C03628=1090.288,180.141,-70.084,176.047,19.774,152.993
C03629=1090.283,179.893,-70.061,176.045,19.773,152.994
C03630=1090.276,179.644,-70.040,176.042,19.772,152.994
C03631=1090.271,179.395,-70.017,176.039,19.771,152.994
C03632=1090.265,179.146,-69.995,176.036,19.769,152.994
C03633=1090.259,178.898,-69.973,176.034,19.768,152.995
C03634=1090.254,178.648,-69.950,176.031,19.767,152.995
C03635=1090.248,178.399,-69.927,176.028,19.766,152.995
C03636=1090.242,178.150,-69.906,176.025,19.765,152.995
C03637=1090.237,177.901,-69.884,176.023,19.764,152.995
C03638=1090.232,177.652,-69.861,176.020,19.763,152.996
C03639=1090.225,177.403,-69.839,176.017,19.762,152.996
C03640=1090.220,177.155,-69.817,176.014,19.761,152.996
C03641=1090.215,176.906,-69.794,176.012,19.760,152.997
C03642=1090.209,176.656,-69.773,176.009,19.759,152.997
C03643=1090.203,176.407,-69.750,176.006,19.758,152.997
C03644=1090.197,176.131,-69.726,176.003,19.756,152.997
C03645=1090.191,175.854,-69.701,176.001,19.755,152.997
C03646=1090.184,175.577,-69.677,175.997,19.753,152.998
C03647=1090.178,175.300,-69.652,175.994,19.752,152.998
C03648=1090.172,175.051,-69.630,175.992,19.751,152.998
C03649=1090.167,174.803,-69.607,175.989,19.750,152.998
C03650=1090.162,174.553,-69.585,175.986,19.749,152.999
C03651=1090.155,174.304,-69.563,175.983,19.748,152.999
C03652=1090.151,174.055,-69.542,175.981,19.747,152.999
C03653=1090.144,173.806,-69.519,175.978,19.746,152.999
C03654=1090.139,173.557,-69.497,175.975,19.745,153.000
C03655=1090.134,173.308,-69.475,175.972,19.744,153.000
C03656=1090.128,173.059,-69.454,175.970,19.742,153.000
C03657=1090.123,172.811,-69.431,175.967,19.741,153.000
C03658=1090.116,172.561,-69.409,175.965,19.740,153.000
C03659=1090.111,172.312,-69.387,175.962,19.739,153.001
C03660=1090.106,172.063,-69.366,175.960,19.738,153.001
C03661=1090.100,171.814,-69.344,175.957,19.737,153.001
C03662=1090.095,171.565,-69.322,175.954,19.736,153.001
C03663=1090.089,171.317,-69.299,175.952,19.734,153.001
C03664=1090.084,171.068,-69.278,175.949,19.733,153.002
C03665=1090.078,170.819,-69.256,175.946,19.732,153.002
C03666=1090.073,170.570,-69.234,175.943,19.731,153.002
C03667=1090.067,170.321,-69.212,175.941,19.730,153.002
C03668=1090.061,170.071,-69.190,175.938,19.729,153.003
C03669=1090.056,169.822,-69.169,175.935,19.728,153.003
C03670=1090.050,169.573,-69.147,175.933,19.726,153.003
C03671=1090.045,169.324,-69.125,175.930,19.725,153.003
C03672=1090.039,169.076,-69.102,175.927,19.724,153.004
C03673=1090.034,168.827,-69.081,175.925,19.722,153.004
C03674=1090.028,168.578,-69.059,175.923,19.722,153.004
C03675=1090.023,168.329,-69.038,175.920,19.720,153.004
C03676=1090.017,168.080,-69.015,175.917,19.719,153.004
C03677=1090.012,167.831,-68.994,175.915,19.718,153.004
C03678=1090.006,167.582,-68.972,175.912,19.717,153.005
C03679=1090.001,167.333,-68.951,175.909,19.716,153.005
C03680=1089.995,167.083,-68.928,175.906,19.715,153.005
C03681=1089.990,166.835,-68.907,175.904,19.713,153.005
C03682=1089.984,166.586,-68.886,175.901,19.712,153.005
C03683=1089.979,166.336,-68.864,175.899,19.711,153.006
C03684=1089.973,166.088,-68.843,175.896,19.710,153.006
C03685=1089.968,165.838,-68.821,175.893,19.708,153.006
C03686=1089.962,165.590,-68.800,175.891,19.707,153.006
C03687=1089.957,165.340,-68.777,175.889,19.707,153.006
C03688=1089.951,165.092,-68.756,175.886,19.705,153.007
C03689=1089.946,164.842,-68.734,175.883,19.704,153.007
C03690=1089.940,164.594,-68.713,175.881,19.702,153.007
C03691=1089.935,164.345,-68.691,175.878,19.701,153.007
C03692=1089.930,164.095,-68.670,175.875,19.700,153.007
C03693=1089.924,163.847,-68.649,175.873,19.699,153.008
C03694=1089.919,163.597,-68.626,175.870,19.697,153.008
C03695=1089.913,163.349,-68.605,175.867,19.696,153.008
C03696=1089.908,163.100,-68.584,175.865,19.695,153.008
C03697=1089.902,162.851,-68.562,175.863,19.694,153.008
C03698=1089.897,162.601,-68.541,175.860,19.693,153.008
C03699=1089.892,162.353,-68.519,175.858,19.692,153.009
C03700=1089.886,162.103,-68.498,175.855,19.690,153.009
C03701=1089.880,161.855,-68.476,175.852,19.689,153.009
C03702=1089.876,161.606,-68.455,175.850,19.688,153.009
C03703=1089.870,161.356,-68.433,175.847,19.687,153.009
C03704=1089.864,161.108,-68.412,175.844,19.685,153.010
C03705=1089.858,160.858,-68.391,175.842,19.684,153.010
C03706=1089.853,160.609,-68.370,175.840,19.683,153.010
C03707=1089.847,160.360,-68.348,175.837,19.682,153.010
C03708=1089.841,160.083,-68.324,175.834,19.680,153.010
C03709=1089.835,159.806,-68.300,175.831,19.679,153.011
C03710=1089.829,159.528,-68.277,175.828,19.678,153.011
C03711=1089.822,159.251,-68.253,175.825,19.677,153.011
C03712=1089.817,159.002,-68.232,175.823,19.675,153.011
C03713=1089.811,158.754,-68.211,175.820,19.674,153.011
C03714=1089.806,158.504,-68.190,175.818,19.673,153.012
C03715=1089.800,158.255,-68.169,175.815,19.672,153.012
C03716=1089.794,158.005,-68.148,175.813,19.671,153.012
C03717=1089.789,157.757,-68.127,175.810,19.670,153.012
C03718=1089.783,157.508,-68.105,175.808,19.668,153.012
C03719=1089.777,157.259,-68.084,175.805,19.667,153.013
C03720=1089.772,157.010,-68.063,175.802,19.666,153.013
C03721=1089.767,156.761,-68.042,175.800,19.664,153.013
C03722=1089.761,156.511,-68.020,175.797,19.663,153.013
C03723=1089.756,156.262,-68.000,175.795,19.662,153.013
C03724=1089.750,156.014,-67.979,175.793,19.661,153.013
C03725=1089.744,155.764,-67.958,175.790,19.660,153.014
C03726=1089.739,155.516,-67.936,175.787,19.658,153.014
C03727=1089.733,155.266,-67.916,175.785,19.657,153.014
C03728=1089.727,155.017,-67.894,175.782,19.656,153.014
C03729=1089.722,154.768,-67.874,175.779,19.655,153.014
C03730=1089.716,154.520,-67.852,175.778,19.654,153.015
C03731=1089.711,154.270,-67.831,175.775,19.653,153.015
C03732=1089.705,154.021,-67.810,175.772,19.651,153.015
C03733=1089.700,153.772,-67.790,175.769,19.650,153.015
C03734=1089.694,153.524,-67.768,175.767,19.649,153.015
C03735=1089.688,153.274,-67.747,175.764,19.648,153.016
C03736=1089.682,153.025,-67.727,175.762,19.647,153.016
C03737=1089.677,152.776,-67.706,175.760,19.646,153.016
C03738=1089.671,152.527,-67.685,175.757,19.644,153.016
C03739=1089.666,152.278,-67.665,175.755,19.642,153.016
C03740=1089.660,152.029,-67.643,175.752,19.641,153.016
C03741=1089.655,151.780,-67.623,175.749,19.640,153.017
C03742=1089.649,151.530,-67.602,175.747,19.639,153.017
C03743=1089.643,151.282,-67.581,175.745,19.638,153.017
C03744=1089.638,151.032,-67.560,175.742,19.636,153.017
C03745=1089.633,150.783,-67.540,175.739,19.635,153.017
C03746=1089.627,150.534,-67.518,175.737,19.634,153.017
C03747=1089.621,150.285,-67.498,175.734,19.633,153.018
C03748=1089.615,150.036,-67.477,175.732,19.632,153.018
C03749=1089.610,149.788,-67.456,175.730,19.630,153.018
C03750=1089.605,149.539,-67.436,175.727,19.629,153.018
C03751=1089.599,149.289,-67.415,175.725,19.628,153.018
C03752=1089.594,149.040,-67.394,175.722,19.626,153.018
C03753=1089.588,148.791,-67.373,175.719,19.625,153.019
C03754=1089.582,148.542,-67.353,175.718,19.624,153.019
C03755=1089.576,148.292,-67.332,175.715,19.623,153.019
C03756=1089.571,148.043,-67.311,175.712,19.622,153.019
C03757=1089.566,147.794,-67.291,175.710,19.620,153.019
C03758=1089.559,147.546,-67.270,175.707,19.619,153.020
C03759=1089.554,147.297,-67.250,175.705,19.618,153.020
C03760=1089.548,147.047,-67.229,175.703,19.616,153.020
C03761=1089.543,146.798,-67.208,175.700,19.615,153.020
C03762=1089.537,146.549,-67.188,175.697,19.614,153.020
C03763=1089.532,146.300,-67.168,175.695,19.613,153.020
C03764=1089.526,146.051,-67.147,175.693,19.612,153.020
C03765=1089.520,145.801,-67.127,175.690,19.610,153.021
C03766=1089.514,145.553,-67.105,175.688,19.609,153.021
C03767=1089.509,145.304,-67.085,175.685,19.608,153.021
C03768=1089.504,145.055,-67.064,175.683,19.606,153.021
C03769=1089.498,144.806,-67.044,175.681,19.606,153.021
C03770=1089.493,144.557,-67.024,175.678,19.604,153.021
C03771=1089.487,144.307,-67.003,175.676,19.603,153.022
C03772=1089.480,144.030,-66.981,175.673,19.601,153.022
C03773=1089.474,143.752,-66.958,175.670,19.600,153.022
C03774=1089.468,143.475,-66.935,175.668,19.599,153.022
C03775=1089.462,143.197,-66.912,175.665,19.597,153.022
C03776=1089.456,142.948,-66.892,175.662,19.596,153.022
C03777=1089.451,142.699,-66.872,175.660,19.594,153.023
C03778=1089.445,142.450,-66.851,175.657,19.593,153.023
C03779=1089.439,142.201,-66.831,175.655,19.591,153.023
C03780=1089.434,141.951,-66.810,175.653,19.591,153.023
C03781=1089.428,141.702,-66.790,175.650,19.589,153.023
C03782=1089.422,141.453,-66.770,175.648,19.588,153.023
C03783=1089.417,141.204,-66.749,175.645,19.586,153.023
C03784=1089.412,140.955,-66.729,175.643,19.585,153.024
C03785=1089.406,140.706,-66.709,175.641,19.584,153.024
C03786=1089.401,140.457,-66.689,175.638,19.583,153.024
C03787=1089.395,140.208,-66.669,175.636,19.581,153.024
C03788=1089.390,139.959,-66.648,175.633,19.580,153.024
C03789=1089.384,139.710,-66.629,175.631,19.579,153.024
C03790=1089.378,139.461,-66.608,175.629,19.578,153.024
C03791=1089.372,139.211,-66.588,175.626,19.576,153.025
C03792=1089.366,138.962,-66.567,175.624,19.575,153.025
C03793=1089.361,138.713,-66.548,175.622,19.574,153.025
C03794=1089.356,138.463,-66.527,175.619,19.573,153.025
C03795=1089.350,138.215,-66.507,175.617,19.571,153.025
C03796=1089.344,137.966,-66.487,175.614,19.570,153.025
C03797=1089.338,137.717,-66.467,175.611,19.568,153.025
C03798=1089.333,137.467,-66.447,175.610,19.567,153.026
C03799=1089.327,137.218,-66.427,175.607,19.566,153.026
C03800=1089.322,136.969,-66.406,175.604,19.564,153.026
C03801=1089.316,136.720,-66.387,175.602,19.563,153.026
C03802=1089.310,136.471,-66.367,175.600,19.562,153.026
C03803=1089.305,136.222,-66.347,175.598,19.560,153.026
C03804=1089.299,135.973,-66.327,175.595,19.559,153.026
C03805=1089.294,135.724,-66.306,175.592,19.558,153.027
C03806=1089.288,135.474,-66.287,175.591,19.557,153.027
C03807=1089.283,135.225,-66.266,175.588,19.555,153.027
C03808=1089.277,134.976,-66.246,175.586,19.554,153.027
C03809=1089.271,134.727,-66.227,175.583,19.552,153.027
C03810=1089.266,134.478,-66.207,175.581,19.551,153.027
C03811=1089.260,134.229,-66.187,175.579,19.550,153.027
C03812=1089.254,133.980,-66.167,175.576,19.548,153.027
C03813=1089.249,133.730,-66.147,175.574,19.547,153.028
C03814=1089.243,133.482,-66.127,175.572,19.546,153.028
C03815=1089.238,133.232,-66.107,175.569,19.545,153.028
C03816=1089.232,132.983,-66.087,175.567,19.543,153.028
C03817=1089.226,132.734,-66.068,175.565,19.542,153.028
C03818=1089.221,132.485,-66.047,175.562,19.541,153.028
C03819=1089.215,132.236,-66.027,175.560,19.539,153.028
C03820=1089.210,131.986,-66.008,175.557,19.537,153.029
C03821=1089.204,131.737,-65.988,175.556,19.536,153.029
C03822=1089.199,131.488,-65.968,175.553,19.535,153.029
C03823=1089.193,131.239,-65.948,175.550,19.534,153.029
C03824=1089.187,130.989,-65.929,175.548,19.532,153.029
C03825=1089.181,130.741,-65.909,175.546,19.531,153.029
C03826=1089.175,130.491,-65.890,175.544,19.530,153.029
C03827=1089.170,130.242,-65.869,175.541,19.528,153.029
C03828=1089.164,129.993,-65.850,175.539,19.527,153.030
C03829=1089.158,129.744,-65.830,175.537,19.526,153.030
C03830=1089.153,129.494,-65.811,175.534,19.524,153.030
C03831=1089.147,129.246,-65.791,175.532,19.523,153.030
C03832=1089.141,128.996,-65.772,175.530,19.522,153.030
C03833=1089.135,128.747,-65.752,175.527,19.521,153.030
C03834=1089.130,128.498,-65.732,175.525,19.519,153.030
C03835=1089.125,128.250,-65.712,175.522,19.518,153.031
C03836=1089.118,127.971,-65.691,175.520,19.516,153.031
C03837=1089.112,127.694,-65.669,175.517,19.515,153.031
C03838=1089.105,127.416,-65.647,175.515,19.513,153.031
C03839=1089.099,127.138,-65.625,175.512,19.512,153.031
C03840=1089.094,126.889,-65.606,175.510,19.511,153.031
C03841=1089.088,126.640,-65.586,175.508,19.509,153.031
C03842=1089.082,126.391,-65.567,175.505,19.507,153.031
C03843=1089.076,126.141,-65.547,175.504,19.506,153.031
C03844=1089.070,125.892,-65.527,175.501,19.505,153.032
C03845=1089.065,125.644,-65.509,175.499,19.503,153.032
C03846=1089.059,125.394,-65.489,175.496,19.502,153.032
C03847=1089.053,125.146,-65.469,175.494,19.501,153.032
C03848=1089.048,124.896,-65.450,175.492,19.499,153.032
C03849=1089.043,124.646,-65.430,175.489,19.498,153.032
C03850=1089.037,124.397,-65.411,175.488,19.497,153.032
C03851=1089.031,124.148,-65.391,175.485,19.495,153.032
C03852=1089.026,123.899,-65.372,175.482,19.494,153.033
C03853=1089.020,123.650,-65.353,175.481,19.493,153.033
C03854=1089.015,123.400,-65.334,175.478,19.491,153.033
C03855=1089.009,123.152,-65.314,175.476,19.489,153.033
C03856=1089.003,122.902,-65.295,175.473,19.488,153.033
C03857=1088.997,122.653,-65.275,175.472,19.487,153.033
C03858=1088.992,122.404,-65.256,175.469,19.485,153.033
C03859=1088.986,122.155,-65.236,175.467,19.484,153.033
C03860=1088.981,121.906,-65.217,175.465,19.483,153.033
C03861=1088.975,121.656,-65.198,175.462,19.481,153.033
C03862=1088.969,121.407,-65.179,175.460,19.480,153.034
C03863=1088.964,121.158,-65.160,175.458,19.479,153.034
C03864=1088.958,120.909,-65.141,175.456,19.477,153.034
C03865=1088.953,120.659,-65.121,175.453,19.475,153.034
C03866=1088.947,120.411,-65.101,175.452,19.474,153.034
C03867=1088.942,120.162,-65.083,175.449,19.472,153.034
C03868=1088.936,119.912,-65.063,175.447,19.471,153.034
C03869=1088.930,119.663,-65.044,175.445,19.470,153.034
C03870=1088.925,119.414,-65.025,175.443,19.468,153.034
C03871=1088.919,119.165,-65.006,175.440,19.466,153.034
C03872=1088.914,118.915,-64.987,175.438,19.465,153.034
C03873=1088.908,118.666,-64.967,175.436,19.464,153.034
C03874=1088.902,118.416,-64.948,175.433,19.462,153.035
C03875=1088.897,118.168,-64.929,175.431,19.460,153.035
C03876=1088.892,117.918,-64.910,175.429,19.459,153.035
C03877=1088.886,117.669,-64.891,175.427,19.458,153.035
C03878=1088.881,117.420,-64.872,175.424,19.456,153.035
C03879=1088.875,117.171,-64.853,175.423,19.455,153.035
C03880=1088.869,116.921,-64.833,175.420,19.453,153.035
C03881=1088.864,116.673,-64.815,175.418,19.452,153.035
C03882=1088.859,116.423,-64.795,175.416,19.451,153.035
C03883=1088.853,116.174,-64.776,175.414,19.449,153.035
C03884=1088.848,115.925,-64.757,175.411,19.447,153.035
C03885=1088.842,115.676,-64.738,175.409,19.446,153.035
C03886=1088.837,115.426,-64.719,175.407,19.445,153.036
C03887=1088.831,115.177,-64.700,175.405,19.443,153.036
C03888=1088.825,114.928,-64.681,175.403,19.442,153.036
C03889=1088.819,114.679,-64.662,175.400,19.440,153.036
C03890=1088.814,114.430,-64.643,175.398,19.438,153.036
C03891=1088.809,114.181,-64.624,175.396,19.437,153.036
C03892=1088.803,113.931,-64.605,175.394,19.435,153.036
C03893=1088.798,113.682,-64.586,175.391,19.434,153.036
C03894=1088.792,113.433,-64.568,175.390,19.432,153.036
C03895=1088.786,113.183,-64.549,175.387,19.431,153.036
C03896=1088.780,112.934,-64.529,175.386,19.430,153.036
C03897=1088.775,112.685,-64.510,175.383,19.428,153.036
C03898=1088.769,112.436,-64.492,175.381,19.426,153.036
C03899=1088.763,112.186,-64.473,175.379,19.425,153.036
C03900=1088.757,111.908,-64.452,175.377,19.424,153.037
C03901=1088.751,111.631,-64.431,175.374,19.422,153.037
C03902=1088.745,111.353,-64.410,175.372,19.420,153.037
C03903=1088.738,111.076,-64.389,175.369,19.419,153.037
C03904=1088.733,110.827,-64.370,175.367,19.417,153.037
C03905=1088.727,110.578,-64.352,175.365,19.416,153.037
C03906=1088.722,110.328,-64.333,175.363,19.414,153.037
C03907=1088.716,110.079,-64.315,175.360,19.413,153.037
C03908=1088.710,109.830,-64.296,175.358,19.412,153.037
C03909=1088.704,109.580,-64.277,175.356,19.410,153.037
C03910=1088.699,109.331,-64.259,175.354,19.408,153.037
C03911=1088.693,109.082,-64.240,175.352,19.407,153.037
C03912=1088.687,108.833,-64.220,175.350,19.405,153.037
C03913=1088.682,108.584,-64.203,175.347,19.403,153.038
C03914=1088.676,108.334,-64.184,175.345,19.402,153.038
C03915=1088.670,108.085,-64.165,175.343,19.400,153.038
C03916=1088.665,107.836,-64.147,175.341,19.399,153.038
C03917=1088.659,107.586,-64.128,175.339,19.398,153.038
C03918=1088.653,107.338,-64.109,175.337,19.396,153.038
C03919=1088.648,107.088,-64.091,175.335,19.395,153.038
C03920=1088.642,106.839,-64.072,175.332,19.393,153.038
C03921=1088.637,106.590,-64.053,175.330,19.391,153.038
C03922=1088.630,106.340,-64.035,175.328,19.390,153.038
C03923=1088.625,106.091,-64.016,175.326,19.388,153.038
C03924=1088.619,105.842,-63.999,175.324,19.387,153.038
C03925=1088.614,105.593,-63.980,175.322,19.386,153.038
C03926=1088.609,105.343,-63.961,175.320,19.384,153.038
C03927=1088.603,105.094,-63.943,175.318,19.383,153.038
C03928=1088.597,104.845,-63.924,175.316,19.381,153.038
C03929=1088.591,104.595,-63.906,175.313,19.379,153.039
C03930=1088.586,104.347,-63.887,175.311,19.378,153.039
C03931=1088.580,104.097,-63.869,175.309,19.376,153.039
C03932=1088.575,103.848,-63.850,175.307,19.375,153.039
C03933=1088.569,103.598,-63.832,175.305,19.373,153.039
C03934=1088.564,103.350,-63.813,175.303,19.371,153.039
C03935=1088.558,103.100,-63.795,175.301,19.370,153.039
C03936=1088.552,102.851,-63.776,175.299,19.368,153.039
C03937=1088.546,102.601,-63.758,175.297,19.367,153.039
C03938=1088.541,102.353,-63.740,175.295,19.365,153.039
C03939=1088.535,102.103,-63.722,175.292,19.364,153.039
C03940=1088.530,101.854,-63.703,175.291,19.362,153.039
C03941=1088.524,101.604,-63.685,175.288,19.361,153.039
C03942=1088.519,101.355,-63.667,175.287,19.359,153.039
C03943=1088.513,101.106,-63.648,175.284,19.358,153.039
C03944=1088.508,100.857,-63.630,175.282,19.356,153.039
C03945=1088.502,100.607,-63.612,175.280,19.355,153.039
C03946=1088.496,100.358,-63.594,175.278,19.353,153.039
C03947=1088.491,100.108,-63.575,175.276,19.352,153.039
C03948=1088.485,99.860,-63.557,175.274,19.350,153.039
C03949=1088.479,99.610,-63.539,175.271,19.348,153.040
C03950=1088.474,99.361,-63.521,175.270,19.347,153.040
C03951=1088.467,99.112,-63.502,175.267,19.345,153.040
C03952=1088.462,98.863,-63.485,175.266,19.344,153.040
C03953=1088.457,98.613,-63.466,175.263,19.342,153.040
C03954=1088.451,98.364,-63.448,175.261,19.341,153.040
C03955=1088.445,98.114,-63.430,175.259,19.339,153.040
C03956=1088.439,97.865,-63.412,175.257,19.337,153.040
C03957=1088.433,97.616,-63.393,175.255,19.336,153.040
C03958=1088.428,97.367,-63.375,175.253,19.334,153.040
C03959=1088.422,97.117,-63.357,175.250,19.332,153.040
C03960=1088.417,96.868,-63.339,175.249,19.331,153.040
C03961=1088.411,96.619,-63.321,175.247,19.329,153.040
C03962=1088.405,96.370,-63.303,175.245,19.328,153.040
C03963=1088.400,96.121,-63.286,175.243,19.326,153.040
C03964=1088.393,95.843,-63.265,175.240,19.324,153.040
C03965=1088.387,95.565,-63.245,175.238,19.323,153.040
C03966=1088.381,95.288,-63.225,175.235,19.321,153.040
C03967=1088.375,95.010,-63.205,175.234,19.319,153.040
C03968=1088.369,94.760,-63.186,175.231,19.318,153.040
C03969=1088.363,94.511,-63.169,175.229,19.316,153.040
C03970=1088.358,94.262,-63.151,175.227,19.315,153.040
C03971=1088.352,94.013,-63.133,175.225,19.313,153.040
C03972=1088.346,93.764,-63.115,175.223,19.312,153.041
C03973=1088.341,93.514,-63.097,175.221,19.310,153.041
C03974=1088.335,93.265,-63.079,175.220,19.308,153.040
C03975=1088.329,93.016,-63.061,175.217,19.307,153.041
C03976=1088.323,92.766,-63.043,175.215,19.305,153.041
C03977=1088.319,92.517,-63.025,175.213,19.303,153.041
C03978=1088.313,92.268,-63.007,175.211,19.301,153.041
C03979=1088.307,92.018,-62.989,175.209,19.300,153.041
C03980=1088.301,91.769,-62.972,175.207,19.298,153.041
C03981=1088.296,91.520,-62.954,175.205,19.297,153.041
C03982=1088.291,91.270,-62.936,175.203,19.295,153.041
C03983=1088.285,91.021,-62.918,175.201,19.293,153.041
C03984=1088.280,90.772,-62.901,175.199,19.292,153.041
C03985=1088.273,90.522,-62.883,175.197,19.290,153.041
C03986=1088.268,90.273,-62.865,175.195,19.289,153.041
C03987=1088.262,90.024,-62.848,175.193,19.287,153.041
C03988=1088.256,89.774,-62.830,175.191,19.286,153.041
C03989=1088.251,89.525,-62.812,175.189,19.284,153.041
C03990=1088.245,89.276,-62.794,175.187,19.282,153.041
C03991=1088.239,89.027,-62.777,175.185,19.281,153.041
C03992=1088.234,88.778,-62.759,175.183,19.279,153.041
C03993=1088.227,88.528,-62.741,175.181,19.278,153.041
C03994=1088.222,88.279,-62.724,175.179,19.276,153.041
C03995=1088.216,88.030,-62.706,175.177,19.274,153.041
C03996=1088.210,87.780,-62.688,175.175,19.273,153.041
C03997=1088.205,87.531,-62.670,175.173,19.271,153.041
C03998=1088.199,87.282,-62.653,175.171,19.269,153.041
C03999=1088.193,87.032,-62.635,175.169,19.268,153.041
C04000=1088.188,86.783,-62.617,175.167,19.266,153.041
C04001=1088.182,86.534,-62.600,175.165,19.264,153.041
C04002=1088.176,86.284,-62.582,175.163,19.263,153.041
C04003=1088.170,86.035,-62.564,175.161,19.261,153.041
C04004=1088.165,85.786,-62.548,175.159,19.259,153.041
C04005=1088.160,85.537,-62.530,175.157,19.258,153.041
C04006=1088.154,85.287,-62.512,175.155,19.256,153.041
C04007=1088.148,85.038,-62.494,175.153,19.254,153.041
C04008=1088.143,84.789,-62.477,175.152,19.253,153.041
C04009=1088.136,84.539,-62.459,175.149,19.251,153.041
C04010=1088.131,84.289,-62.442,175.148,19.250,153.041
C04011=1088.126,84.040,-62.425,175.145,19.248,153.041
C04012=1088.120,83.791,-62.407,175.143,19.246,153.041
C04013=1088.114,83.542,-62.389,175.141,19.245,153.041
C04014=1088.109,83.292,-62.371,175.139,19.243,153.041
C04015=1088.103,83.043,-62.355,175.138,19.241,153.041
C04016=1088.097,82.794,-62.338,175.135,19.239,153.041
C04017=1088.091,82.544,-62.320,175.134,19.238,153.041
C04018=1088.085,82.295,-62.302,175.131,19.236,153.041
C04019=1088.080,82.046,-62.285,175.130,19.234,153.041
C04020=1088.075,81.797,-62.268,175.128,19.232,153.041
C04021=1088.069,81.548,-62.250,175.126,19.231,153.041
C04022=1088.063,81.298,-62.232,175.124,19.229,153.041
C04023=1088.058,81.048,-62.215,175.122,19.228,153.041
C04024=1088.052,80.799,-62.198,175.120,19.226,153.041
C04025=1088.047,80.550,-62.180,175.118,19.224,153.041
C04026=1088.041,80.301,-62.164,175.116,19.222,153.041
C04027=1088.035,80.051,-62.146,175.114,19.221,153.041
C04028=1088.029,79.774,-62.126,175.112,19.219,153.041
C04029=1088.023,79.496,-62.108,175.110,19.217,153.041
C04030=1088.016,79.218,-62.088,175.108,19.215,153.041
C04031=1088.010,78.941,-62.069,175.105,19.213,153.041
C04032=1088.005,78.692,-62.052,175.104,19.212,153.041
C04033=1087.999,78.442,-62.035,175.102,19.210,153.041
C04034=1087.994,78.193,-62.017,175.100,19.209,153.041
C04035=1087.987,77.944,-62.000,175.098,19.206,153.041
C04036=1087.982,77.694,-61.983,175.096,19.205,153.041
C04037=1087.976,77.445,-61.965,175.094,19.203,153.041
C04038=1087.970,77.196,-61.949,175.092,19.201,153.041
C04039=1087.965,76.947,-61.932,175.090,19.199,153.041
C04040=1087.959,76.696,-61.914,175.088,19.198,153.041
C04041=1087.953,76.447,-61.897,175.086,19.196,153.041
C04042=1087.948,76.198,-61.881,175.085,19.195,153.041
C04043=1087.942,75.949,-61.863,175.082,19.193,153.041
C04044=1087.936,75.700,-61.845,175.081,19.191,153.041
C04045=1087.931,75.451,-61.829,175.078,19.190,153.041
C04046=1087.924,75.201,-61.811,175.077,19.188,153.041
C04047=1087.919,74.951,-61.794,175.075,19.186,153.041
C04048=1087.913,74.702,-61.777,175.073,19.185,153.041
C04049=1087.908,74.453,-61.761,175.071,19.183,153.041
C04050=1087.903,74.203,-61.744,175.069,19.181,153.041
C04051=1087.896,73.954,-61.727,175.067,19.179,153.041
C04052=1087.891,73.705,-61.710,175.066,19.178,153.041
C04053=1087.886,73.456,-61.692,175.063,19.176,153.041
C04054=1087.879,73.206,-61.676,175.062,19.174,153.041
C04055=1087.873,72.957,-61.658,175.060,19.172,153.041
C04056=1087.868,72.707,-61.641,175.058,19.171,153.041
C04057=1087.862,72.458,-61.625,175.056,19.169,153.041
C04058=1087.857,72.209,-61.608,175.054,19.167,153.041
C04059=1087.851,71.959,-61.591,175.052,19.165,153.041
C04060=1087.845,71.710,-61.574,175.051,19.164,153.041
C04061=1087.840,71.460,-61.557,175.048,19.162,153.041
C04062=1087.834,71.211,-61.541,175.047,19.160,153.041
C04063=1087.829,70.962,-61.523,175.044,19.159,153.041
C04064=1087.823,70.713,-61.507,175.043,19.157,153.041
C04065=1087.817,70.463,-61.490,175.041,19.155,153.041
C04066=1087.812,70.214,-61.472,175.039,19.154,153.041
C04067=1087.805,69.964,-61.456,175.037,19.152,153.041
C04068=1087.800,69.714,-61.439,175.035,19.150,153.041
C04069=1087.794,69.466,-61.422,175.033,19.148,153.041
C04070=1087.789,69.216,-61.405,175.032,19.147,153.041
C04071=1087.783,68.967,-61.389,175.029,19.144,153.041
C04072=1087.777,68.718,-61.371,175.028,19.143,153.041
C04073=1087.771,68.468,-61.355,175.026,19.141,153.041
C04074=1087.766,68.219,-61.338,175.024,19.139,153.041
C04075=1087.760,67.969,-61.322,175.022,19.137,153.041
C04076=1087.755,67.720,-61.304,175.021,19.136,153.041
C04077=1087.749,67.471,-61.288,175.018,19.134,153.041
C04078=1087.743,67.221,-61.271,175.017,19.133,153.041
C04079=1087.738,66.972,-61.255,175.014,19.131,153.041
C04080=1087.732,66.722,-61.238,175.013,19.129,153.041
C04081=1087.726,66.473,-61.221,175.011,19.127,153.041
C04082=1087.720,66.224,-61.205,175.009,19.126,153.041
C04083=1087.715,65.974,-61.188,175.007,19.124,153.041
C04084=1087.709,65.725,-61.172,175.005,19.122,153.041
C04085=1087.704,65.475,-61.155,175.003,19.120,153.041
C04086=1087.697,65.227,-61.138,175.002,19.119,153.041
C04087=1087.692,64.977,-61.121,174.999,19.116,153.041
C04088=1087.686,64.728,-61.105,174.998,19.115,153.041
C04089=1087.680,64.478,-61.089,174.996,19.113,153.041
C04090=1087.675,64.229,-61.072,174.994,19.111,153.041
C04091=1087.669,63.979,-61.055,174.993,19.110,153.040
C04092=1087.662,63.701,-61.037,174.990,19.108,153.040
C04093=1087.655,63.424,-61.019,174.988,19.106,153.040
C04094=1087.649,63.146,-61.000,174.986,19.104,153.040
C04095=1087.643,62.869,-60.982,174.984,19.102,153.040
C04096=1087.637,62.620,-60.966,174.982,19.100,153.040
C04097=1087.631,62.370,-60.949,174.981,19.099,153.040
C04098=1087.626,62.121,-60.932,174.978,19.097,153.040
C04099=1087.620,61.871,-60.916,174.977,19.095,153.040
C04100=1087.614,61.622,-60.900,174.975,19.093,153.040
C04101=1087.608,61.373,-60.884,174.973,19.092,153.040
C04102=1087.603,61.123,-60.867,174.971,19.090,153.040
C04103=1087.597,60.874,-60.851,174.970,19.088,153.040
C04104=1087.591,60.624,-60.834,174.968,19.086,153.040
C04105=1087.585,60.375,-60.818,174.966,19.084,153.040
C04106=1087.579,60.125,-60.802,174.964,19.083,153.040
C04107=1087.574,59.876,-60.785,174.962,19.081,153.040
C04108=1087.568,59.626,-60.769,174.961,19.079,153.040
C04109=1087.562,59.377,-60.752,174.958,19.077,153.040
C04110=1087.556,59.128,-60.736,174.957,19.076,153.040
C04111=1087.550,58.878,-60.720,174.955,19.074,153.040
C04112=1087.545,58.629,-60.703,174.953,19.072,153.040
C04113=1087.539,58.379,-60.687,174.951,19.070,153.040
C04114=1087.533,58.130,-60.671,174.949,19.069,153.040
C04115=1087.527,57.881,-60.654,174.948,19.067,153.040
C04116=1087.521,57.631,-60.638,174.946,19.065,153.040
C04117=1087.515,57.382,-60.622,174.944,19.064,153.040
C04118=1087.510,57.132,-60.605,174.942,19.061,153.040
C04119=1087.504,56.883,-60.589,174.941,19.060,153.040
C04120=1087.499,56.634,-60.574,174.938,19.058,153.040
C04121=1087.493,56.384,-60.557,174.937,19.056,153.040
C04122=1087.487,56.135,-60.541,174.935,19.054,153.040
C04123=1087.481,55.886,-60.525,174.933,19.053,153.040
C04124=1087.475,55.636,-60.508,174.932,19.051,153.040
C04125=1087.469,55.387,-60.492,174.929,19.049,153.040
C04126=1087.464,55.137,-60.475,174.928,19.048,153.040
C04127=1087.458,54.887,-60.460,174.926,19.046,153.040
C04128=1087.452,54.638,-60.444,174.925,19.044,153.039
C04129=1087.447,54.389,-60.428,174.922,19.042,153.039
C04130=1087.441,54.140,-60.411,174.921,19.040,153.039
C04131=1087.435,53.891,-60.395,174.919,19.038,153.039
C04132=1087.429,53.641,-60.380,174.917,19.037,153.039
C04133=1087.423,53.391,-60.363,174.916,19.035,153.039
C04134=1087.418,53.142,-60.347,174.913,19.033,153.039
C04135=1087.413,52.893,-60.331,174.912,19.031,153.039
C04136=1087.407,52.643,-60.315,174.910,19.029,153.039
C04137=1087.401,52.394,-60.299,174.908,19.027,153.039
C04138=1087.395,52.144,-60.283,174.906,19.025,153.039
C04139=1087.389,51.895,-60.266,174.905,19.024,153.039
C04140=1087.384,51.645,-60.251,174.903,19.022,153.039
C04141=1087.378,51.396,-60.235,174.901,19.020,153.039
C04142=1087.372,51.147,-60.219,174.900,19.019,153.039
C04143=1087.367,50.897,-60.203,174.898,19.016,153.039
C04144=1087.361,50.648,-60.187,174.896,19.015,153.039
C04145=1087.355,50.398,-60.171,174.894,19.013,153.039
C04146=1087.350,50.149,-60.155,174.892,19.011,153.039
C04147=1087.345,49.899,-60.139,174.891,19.010,153.038
C04148=1087.339,49.650,-60.122,174.889,19.007,153.038
C04149=1087.333,49.400,-60.107,174.887,19.005,153.038
C04150=1087.328,49.152,-60.091,174.885,19.003,153.038
C04151=1087.322,48.902,-60.075,174.884,19.002,153.038
C04152=1087.316,48.652,-60.059,174.881,19.000,153.038
C04153=1087.310,48.403,-60.043,174.880,18.998,153.038
C04154=1087.305,48.154,-60.028,174.879,18.996,153.038
C04155=1087.299,47.904,-60.011,174.877,18.994,153.038
C04156=1087.292,47.626,-59.994,174.875,18.993,153.038
C04157=1087.287,47.348,-59.976,174.873,18.991,153.038
C04158=1087.281,47.070,-59.959,174.871,18.988,153.038
C04159=1087.274,46.793,-59.941,174.869,18.986,153.038
C04160=1087.268,46.543,-59.925,174.867,18.985,153.038
C04161=1087.262,46.294,-59.909,174.866,18.982,153.038
C04162=1087.257,46.044,-59.894,174.864,18.980,153.038
C04163=1087.251,45.795,-59.878,174.862,18.979,153.037
C04164=1087.245,45.545,-59.862,174.860,18.977,153.037
C04165=1087.240,45.296,-59.846,174.859,18.975,153.037
C04166=1087.234,45.047,-59.831,174.857,18.973,153.037
C04167=1087.228,44.797,-59.814,174.855,18.971,153.037
C04168=1087.223,44.548,-59.799,174.854,18.969,153.037
C04169=1087.217,44.299,-59.783,174.852,18.967,153.037
C04170=1087.212,44.049,-59.767,174.850,18.966,153.037
C04171=1087.206,43.800,-59.752,174.849,18.964,153.037
C04172=1087.201,43.550,-59.736,174.847,18.962,153.037
C04173=1087.195,43.300,-59.720,174.845,18.960,153.037
C04174=1087.189,43.051,-59.704,174.843,18.958,153.037
C04175=1087.183,42.802,-59.690,174.841,18.956,153.037
C04176=1087.177,42.552,-59.673,174.840,18.955,153.037
C04177=1087.172,42.302,-59.658,174.838,18.952,153.037
C04178=1087.167,42.054,-59.642,174.837,18.951,153.036
C04179=1087.161,41.804,-59.626,174.834,18.949,153.036
C04180=1087.154,41.554,-59.611,174.833,18.947,153.036
C04181=1087.149,41.305,-59.596,174.831,18.946,153.036
C04182=1087.143,41.055,-59.580,174.829,18.943,153.036
C04183=1087.138,40.806,-59.564,174.828,18.942,153.036
C04184=1087.132,40.557,-59.549,174.826,18.940,153.036
C04185=1087.126,40.307,-59.534,174.824,18.938,153.036
C04186=1087.120,40.057,-59.518,174.823,18.936,153.036
C04187=1087.115,39.809,-59.502,174.821,18.934,153.036
C04188=1087.109,39.559,-59.487,174.819,18.932,153.036
C04189=1087.103,39.309,-59.472,174.817,18.930,153.036
C04190=1087.098,39.060,-59.456,174.816,18.928,153.036
C04191=1087.092,38.810,-59.440,174.814,18.927,153.036
C04192=1087.086,38.560,-59.425,174.812,18.925,153.036
C04193=1087.080,38.312,-59.409,174.811,18.923,153.036
C04194=1087.075,38.062,-59.394,174.809,18.921,153.035
C04195=1087.070,37.813,-59.379,174.807,18.919,153.035
C04196=1087.064,37.563,-59.363,174.806,18.918,153.035
C04197=1087.057,37.314,-59.348,174.804,18.916,153.035
C04198=1087.052,37.065,-59.332,174.802,18.914,153.035
C04199=1087.046,36.815,-59.317,174.801,18.912,153.035
C04200=1087.040,36.565,-59.302,174.799,18.910,153.035
C04201=1087.035,36.316,-59.287,174.797,18.908,153.035
C04202=1087.029,36.067,-59.271,174.795,18.906,153.035
C04203=1087.023,35.817,-59.256,174.794,18.904,153.035
C04204=1087.017,35.568,-59.241,174.792,18.903,153.035
C04205=1087.011,35.318,-59.225,174.790,18.901,153.035
C04206=1087.006,35.068,-59.210,174.789,18.899,153.035
C04207=1087.000,34.819,-59.195,174.787,18.897,153.035
C04208=1086.994,34.569,-59.179,174.785,18.895,153.035
C04209=1086.988,34.321,-59.164,174.784,18.894,153.035
C04210=1086.983,34.071,-59.149,174.781,18.892,153.035
C04211=1086.976,33.821,-59.134,174.780,18.890,153.034
C04212=1086.971,33.572,-59.119,174.779,18.888,153.034
C04213=1086.966,33.322,-59.103,174.777,18.886,153.034
C04214=1086.959,33.073,-59.088,174.775,18.884,153.034
C04215=1086.954,32.823,-59.072,174.774,18.882,153.034
C04216=1086.948,32.574,-59.058,174.772,18.880,153.034
C04217=1086.942,32.324,-59.042,174.770,18.879,153.034
C04218=1086.936,32.075,-59.027,174.768,18.876,153.034
C04219=1086.931,31.825,-59.012,174.767,18.875,153.034
C04220=1086.922,31.451,-58.990,174.765,18.872,153.034
C04221=1086.914,31.077,-58.967,174.762,18.869,153.034
C04222=1086.905,30.702,-58.944,174.759,18.866,153.034
C04223=1086.896,30.328,-58.921,174.757,18.863,153.033
C04224=1086.890,30.078,-58.906,174.756,18.862,153.033
C04225=1086.885,29.829,-58.891,174.753,18.860,153.033
C04226=1086.879,29.579,-58.876,174.752,18.858,153.033
C04227=1086.873,29.330,-58.861,174.750,18.856,153.033
C04228=1086.868,29.080,-58.846,174.748,18.854,153.033
C04229=1086.862,28.831,-58.831,174.747,18.852,153.033
C04230=1086.856,28.581,-58.816,174.745,18.850,153.033
C04231=1086.850,28.332,-58.801,174.743,18.849,153.033
C04232=1086.845,28.082,-58.785,174.742,18.847,153.033
C04233=1086.839,27.833,-58.771,174.740,18.844,153.033
C04234=1086.833,27.584,-58.756,174.739,18.843,153.033
C04235=1086.828,27.334,-58.741,174.737,18.841,153.033
C04236=1086.821,27.084,-58.726,174.735,18.839,153.032
C04237=1086.816,26.835,-58.711,174.734,18.837,153.032
C04238=1086.810,26.585,-58.696,174.732,18.836,153.032
C04239=1086.804,26.336,-58.682,174.730,18.833,153.032
C04240=1086.799,26.086,-58.666,174.729,18.832,153.032
C04241=1086.793,25.837,-58.652,174.727,18.830,153.032
C04242=1086.786,25.588,-58.637,174.725,18.828,153.032
C04243=1086.781,25.338,-58.622,174.724,18.826,153.032
C04244=1086.775,25.088,-58.607,174.723,18.825,153.032
C04245=1086.770,24.839,-58.593,174.720,18.822,153.032
C04246=1086.764,24.589,-58.577,174.719,18.820,153.032
C04247=1086.758,24.340,-58.563,174.718,18.819,153.032
C04248=1086.752,24.091,-58.548,174.715,18.817,153.032
C04249=1086.747,23.841,-58.532,174.714,18.815,153.031
C04250=1086.741,23.591,-58.518,174.713,18.813,153.031
C04251=1086.735,23.342,-58.504,174.710,18.811,153.031
C04252=1086.729,23.092,-58.488,174.709,18.809,153.031
C04253=1086.723,22.843,-58.474,174.708,18.808,153.031
C04254=1086.717,22.594,-58.459,174.706,18.806,153.031
C04255=1086.712,22.344,-58.445,174.704,18.804,153.031
C04256=1086.707,22.095,-58.430,174.703,18.802,153.031
C04257=1086.700,21.845,-58.415,174.701,18.800,153.031
C04258=1086.694,21.596,-58.400,174.700,18.798,153.031
C04259=1086.689,21.346,-58.385,174.698,18.796,153.031
C04260=1086.683,21.097,-58.371,174.696,18.794,153.031
C04261=1086.677,20.847,-58.356,174.695,18.792,153.031
C04262=1086.671,20.598,-58.341,174.693,18.791,153.030
C04263=1086.666,20.348,-58.327,174.691,18.789,153.030
C04264=1086.656,19.946,-58.303,174.688,18.786,153.030
C04265=1086.647,19.543,-58.279,174.686,18.783,153.030
C04266=1086.638,19.141,-58.256,174.683,18.779,153.030
C04267=1086.628,18.738,-58.233,174.681,18.776,153.030
C04268=1086.623,18.489,-58.217,174.679,18.775,153.030
C04269=1086.617,18.240,-58.202,174.678,18.773,153.030
C04270=1086.611,17.990,-58.189,174.676,18.771,153.030
C04271=1086.605,17.740,-58.174,174.674,18.769,153.030
C04272=1086.599,17.491,-58.160,174.673,18.768,153.030
C04273=1086.594,17.242,-58.145,174.671,18.765,153.029
C04274=1086.588,16.992,-58.130,174.669,18.764,153.029
C04275=1086.583,16.742,-58.116,174.668,18.761,153.029
C04276=1086.576,16.493,-58.101,174.666,18.759,153.029
C04277=1086.571,16.243,-58.087,174.665,18.758,153.029
C04278=1086.565,15.994,-58.072,174.663,18.756,153.029
C04279=1086.558,15.744,-58.057,174.661,18.754,153.029
C04280=1086.552,15.468,-58.042,174.660,18.752,153.029
C04281=1086.546,15.192,-58.025,174.658,18.750,153.029
C04282=1086.539,14.915,-58.010,174.656,18.748,153.029
C04283=1086.534,14.638,-57.994,174.654,18.746,153.029
C04284=1086.528,14.389,-57.979,174.653,18.744,153.029
C04285=1086.522,14.140,-57.964,174.652,18.742,153.028
C04286=1086.516,13.890,-57.950,174.649,18.740,153.028
C04287=1086.510,13.641,-57.936,174.648,18.738,153.028
C04288=1086.505,13.391,-57.922,174.646,18.737,153.028
C04289=1086.498,13.141,-57.907,174.644,18.734,153.028
C04290=1086.492,12.892,-57.894,174.643,18.733,153.028
C04291=1086.486,12.643,-57.879,174.642,18.731,153.028
C04292=1086.480,12.393,-57.865,174.640,18.729,153.028
C04293=1086.475,12.143,-57.851,174.638,18.727,153.028
C04294=1086.468,11.894,-57.836,174.637,18.726,153.028
C04295=1086.463,11.644,-57.822,174.636,18.724,153.028
C04296=1086.457,11.395,-57.807,174.633,18.721,153.028
C04297=1086.451,11.145,-57.793,174.632,18.720,153.028
C04298=1086.445,10.896,-57.779,174.630,18.718,153.028
C04299=1086.440,10.646,-57.765,174.628,18.716,153.027
C04300=1086.434,10.396,-57.751,174.627,18.714,153.027
C04301=1086.428,10.147,-57.736,174.626,18.713,153.027
C04302=1086.422,9.897,-57.722,174.624,18.711,153.027
C04303=1086.416,9.648,-57.707,174.622,18.709,153.027
C04304=1086.410,9.399,-57.694,174.621,18.707,153.027
C04305=1086.404,9.149,-57.680,174.619,18.705,153.027
C04306=1086.399,8.900,-57.665,174.617,18.703,153.027
C04307=1086.393,8.650,-57.651,174.616,18.701,153.027
C04308=1086.387,8.400,-57.637,174.615,18.699,153.027
C04309=1086.381,8.151,-57.623,174.612,18.697,153.027
C04310=1086.375,7.901,-57.609,174.611,18.696,153.027
C04311=1086.370,7.651,-57.595,174.610,18.694,153.026
C04312=1086.364,7.402,-57.580,174.608,18.692,153.026
C04313=1086.358,7.153,-57.567,174.606,18.690,153.026
C04314=1086.352,6.903,-57.553,174.605,18.688,153.026
C04315=1086.346,6.654,-57.538,174.603,18.687,153.026
C04316=1086.340,6.404,-57.524,174.601,18.685,153.026
C04317=1086.335,6.155,-57.510,174.600,18.682,153.026
C04318=1086.329,5.904,-57.496,174.599,18.681,153.026
C04319=1086.323,5.656,-57.481,174.597,18.679,153.026
C04320=1086.318,5.406,-57.468,174.595,18.677,153.026
C04321=1086.311,5.157,-57.454,174.594,18.675,153.026
C04322=1086.305,4.906,-57.440,174.593,18.673,153.026
C04323=1086.299,4.657,-57.426,174.591,18.672,153.025
C04324=1086.294,4.408,-57.412,174.589,18.670,153.025
C04325=1086.289,4.158,-57.398,174.588,18.668,153.025
C04326=1086.282,3.908,-57.384,174.586,18.666,153.025
C04327=1086.276,3.659,-57.370,174.584,18.664,153.025
C04328=1086.270,3.410,-57.356,174.583,18.662,153.025
C04329=1086.265,3.160,-57.342,174.581,18.660,153.025
C04330=1086.259,2.911,-57.328,174.580,18.659,153.025
C04331=1086.253,2.660,-57.314,174.578,18.656,153.025
C04332=1086.248,2.411,-57.300,174.576,18.655,153.025
C04333=1086.241,2.162,-57.286,174.575,18.653,153.025
C04334=1086.236,1.913,-57.272,174.573,18.651,153.025
C04335=1086.230,1.663,-57.258,174.572,18.649,153.025
C04336=1086.225,1.413,-57.244,174.570,18.647,153.024
C04337=1086.219,1.163,-57.230,174.569,18.645,153.024
C04338=1086.213,0.914,-57.217,174.567,18.643,153.024
C04339=1086.207,0.664,-57.203,174.566,18.641,153.024
C04340=1086.202,0.415,-57.189,174.564,18.640,153.024
C04341=1086.196,0.165,-57.175,174.563,18.638,153.024
C04342=1086.190,-0.084,-57.161,174.561,18.636,153.024
C04343=1086.184,-0.333,-57.147,174.559,18.634,153.024
C04344=1086.178,-0.608,-57.133,174.558,18.632,153.024
C04345=1086.171,-0.882,-57.117,174.556,18.630,153.024
C04346=1086.166,-1.157,-57.102,174.555,18.628,153.024
C04347=1086.159,-1.431,-57.087,174.553,18.625,153.023
C04348=1086.153,-1.681,-57.073,174.551,18.624,153.023
C04349=1086.148,-1.930,-57.059,174.550,18.622,153.023
C04350=1086.143,-2.180,-57.045,174.548,18.620,153.023
C04351=1086.136,-2.430,-57.032,174.546,18.618,153.023
C04352=1086.130,-2.679,-57.018,174.545,18.616,153.023
C04353=1086.125,-2.929,-57.004,174.544,18.615,153.023
C04354=1086.119,-3.179,-56.990,174.542,18.613,153.023
C04355=1086.113,-3.428,-56.977,174.540,18.610,153.023
C04356=1086.108,-3.677,-56.963,174.539,18.609,153.023
C04357=1086.101,-3.927,-56.950,174.537,18.607,153.023
C04358=1086.096,-4.176,-56.936,174.536,18.605,153.022
C04359=1086.089,-4.426,-56.922,174.534,18.603,153.022
C04360=1086.084,-4.676,-56.908,174.533,18.602,153.022
C04361=1086.078,-4.925,-56.894,174.531,18.600,153.022
C04362=1086.072,-5.175,-56.881,174.529,18.598,153.022
C04363=1086.066,-5.424,-56.867,174.528,18.596,153.022
C04364=1086.060,-5.674,-56.854,174.526,18.595,153.022
C04365=1086.055,-5.923,-56.840,174.525,18.592,153.022
C04366=1086.049,-6.172,-56.827,174.523,18.590,153.022
C04367=1086.043,-6.423,-56.813,174.522,18.589,153.022
C04368=1086.037,-6.673,-56.800,174.520,18.587,153.022
C04369=1086.031,-6.922,-56.786,174.519,18.585,153.022
C04370=1086.025,-7.171,-56.773,174.517,18.583,153.022
C04371=1086.019,-7.421,-56.759,174.516,18.581,153.021
C04372=1086.013,-7.670,-56.746,174.514,18.580,153.021
C04373=1086.008,-7.920,-56.732,174.513,18.578,153.021
C04374=1086.001,-8.169,-56.719,174.510,18.576,153.021
C04375=1085.996,-8.419,-56.706,174.509,18.574,153.021
C04376=1085.990,-8.668,-56.692,174.508,18.572,153.021
C04377=1085.984,-8.919,-56.678,174.506,18.571,153.021
C04378=1085.978,-9.168,-56.665,174.504,18.568,153.021
C04379=1085.972,-9.418,-56.651,174.503,18.567,153.021
C04380=1085.966,-9.667,-56.638,174.502,18.565,153.021
C04381=1085.961,-9.917,-56.624,174.500,18.563,153.021
C04382=1085.955,-10.166,-56.611,174.498,18.561,153.021
C04383=1085.949,-10.416,-56.597,174.497,18.559,153.021
C04384=1085.943,-10.665,-56.584,174.496,18.557,153.020
C04385=1085.937,-10.915,-56.572,174.494,18.556,153.020
C04386=1085.932,-11.165,-56.558,174.493,18.554,153.020
C04387=1085.925,-11.414,-56.544,174.491,18.552,153.020
C04388=1085.920,-11.663,-56.531,174.489,18.550,153.020
C04389=1085.914,-11.913,-56.518,174.488,18.549,153.020
C04390=1085.909,-12.163,-56.504,174.487,18.547,153.020
C04391=1085.902,-12.412,-56.491,174.484,18.545,153.020
C04392=1085.897,-12.662,-56.478,174.483,18.543,153.020
C04393=1085.891,-12.912,-56.464,174.482,18.541,153.020
C04394=1085.885,-13.161,-56.451,174.480,18.539,153.020
C04395=1085.879,-13.410,-56.437,174.478,18.537,153.020
C04396=1085.873,-13.660,-56.425,174.477,18.535,153.020
C04397=1085.868,-13.910,-56.411,174.476,18.534,153.020
C04398=1085.862,-14.159,-56.398,174.474,18.532,153.019
C04399=1085.857,-14.409,-56.384,174.473,18.530,153.019
C04400=1085.850,-14.659,-56.371,174.471,18.528,153.019
C04401=1085.844,-14.908,-56.358,174.469,18.527,153.019
C04402=1085.839,-15.158,-56.345,174.468,18.524,153.019
C04403=1085.833,-15.407,-56.332,174.467,18.523,153.019
C04404=1085.827,-15.657,-56.319,174.464,18.521,153.019
C04405=1085.821,-15.907,-56.306,174.463,18.519,153.019
C04406=1085.815,-16.156,-56.292,174.462,18.517,153.019
C04407=1085.809,-16.406,-56.279,174.460,18.516,153.019
C04408=1085.803,-16.679,-56.265,174.458,18.514,153.019
C04409=1085.797,-16.951,-56.251,174.457,18.512,153.019
C04410=1085.790,-17.224,-56.235,174.456,18.510,153.019
C04411=1085.784,-17.497,-56.221,174.453,18.508,153.019
C04412=1085.778,-17.747,-56.209,174.452,18.506,153.018
C04413=1085.771,-17.996,-56.195,174.451,18.504,153.018
C04414=1085.766,-18.246,-56.183,174.449,18.503,153.018
C04415=1085.759,-18.495,-56.170,174.447,18.501,153.018
C04416=1085.754,-18.745,-56.156,174.446,18.499,153.018
C04417=1085.748,-18.995,-56.143,174.444,18.497,153.018
C04418=1085.742,-19.244,-56.131,174.443,18.496,153.018
C04419=1085.736,-19.494,-56.117,174.442,18.494,153.018
C04420=1085.731,-19.744,-56.104,174.440,18.491,153.018
C04421=1085.724,-19.993,-56.091,174.438,18.490,153.018
C04422=1085.719,-20.243,-56.078,174.437,18.488,153.018
C04423=1085.713,-20.492,-56.065,174.435,18.487,153.018
C04424=1085.707,-20.741,-56.053,174.434,18.485,153.018
C04425=1085.701,-20.991,-56.040,174.432,18.483,153.018
C04426=1085.696,-21.241,-56.026,174.430,18.481,153.017
C04427=1085.689,-21.490,-56.013,174.429,18.479,153.017
C04428=1085.683,-21.740,-56.001,174.428,18.478,153.017
C04429=1085.677,-21.989,-55.987,174.426,18.476,153.017
C04430=1085.671,-22.239,-55.975,174.424,18.474,153.017
C04431=1085.666,-22.489,-55.961,174.423,18.472,153.017
C04432=1085.660,-22.739,-55.948,174.422,18.470,153.017
C04433=1085.654,-22.989,-55.936,174.420,18.469,153.017
C04434=1085.648,-23.237,-55.923,174.419,18.467,153.017
C04435=1085.643,-23.487,-55.910,174.417,18.465,153.017
C04436=1085.636,-23.736,-55.897,174.415,18.463,153.017
C04437=1085.631,-23.986,-55.884,174.414,18.462,153.017
C04438=1085.625,-24.236,-55.871,174.413,18.460,153.017
C04439=1085.619,-24.486,-55.858,174.411,18.458,153.016
C04440=1085.613,-24.735,-55.846,174.409,18.456,153.016
C04441=1085.607,-24.985,-55.833,174.408,18.454,153.016
C04442=1085.602,-25.234,-55.820,174.406,18.453,153.016
C04443=1085.596,-25.484,-55.808,174.405,18.451,153.016
C04444=1085.591,-25.734,-55.794,174.404,18.449,153.016
C04445=1085.584,-25.983,-55.781,174.402,18.448,153.016
C04446=1085.578,-26.233,-55.769,174.400,18.446,153.016
C04447=1085.573,-26.483,-55.756,174.399,18.443,153.016
C04448=1085.567,-26.732,-55.743,174.397,18.442,153.016
C04449=1085.561,-26.981,-55.731,174.396,18.440,153.016
C04450=1085.555,-27.231,-55.718,174.395,18.439,153.016
C04451=1085.549,-27.481,-55.705,174.393,18.436,153.016
C04452=1085.543,-27.730,-55.692,174.391,18.435,153.016
C04453=1085.537,-27.980,-55.680,174.390,18.433,153.016
C04454=1085.531,-28.230,-55.667,174.388,18.432,153.016
C04455=1085.526,-28.479,-55.654,174.387,18.430,153.016
C04456=1085.520,-28.729,-55.642,174.385,18.428,153.015
C04457=1085.514,-28.979,-55.629,174.383,18.426,153.015
C04458=1085.508,-29.228,-55.617,174.382,18.424,153.015
C04459=1085.502,-29.478,-55.603,174.381,18.423,153.015
C04460=1085.496,-29.728,-55.591,174.379,18.421,153.015
C04461=1085.489,-29.977,-55.579,174.378,18.420,153.015
C04462=1085.484,-30.226,-55.567,174.376,18.418,153.015
C04463=1085.478,-30.476,-55.554,174.374,18.416,153.015
C04464=1085.472,-30.726,-55.541,174.373,18.414,153.015
C04465=1085.466,-30.975,-55.528,174.372,18.412,153.015
C04466=1085.460,-31.225,-55.516,174.370,18.411,153.015
C04467=1085.454,-31.474,-55.503,174.369,18.409,153.015
C04468=1085.449,-31.724,-55.491,174.368,18.407,153.015
C04469=1085.443,-31.974,-55.478,174.365,18.405,153.015
C04470=1085.436,-32.223,-55.465,174.364,18.404,153.015
C04471=1085.431,-32.473,-55.453,174.362,18.402,153.015
C04472=1085.424,-32.745,-55.439,174.361,18.401,153.015
C04473=1085.418,-33.017,-55.426,174.359,18.398,153.014
C04474=1085.411,-33.289,-55.412,174.358,18.396,153.014
C04475=1085.405,-33.561,-55.398,174.356,18.395,153.014
C04476=1085.399,-33.811,-55.386,174.355,18.393,153.014
C04477=1085.393,-34.060,-55.374,174.353,18.391,153.014
C04478=1085.387,-34.310,-55.361,174.351,18.389,153.014
C04479=1085.382,-34.560,-55.349,174.350,18.388,153.014
C04480=1085.376,-34.809,-55.337,174.349,18.386,153.014
C04481=1085.370,-35.059,-55.324,174.347,18.385,153.014
C04482=1085.364,-35.309,-55.311,174.346,18.383,153.014
C04483=1085.358,-35.558,-55.299,174.344,18.381,153.014
C04484=1085.352,-35.807,-55.287,174.342,18.379,153.014
C04485=1085.346,-36.057,-55.274,174.341,18.377,153.014
C04486=1085.340,-36.306,-55.262,174.339,18.376,153.014
C04487=1085.335,-36.556,-55.249,174.338,18.374,153.014
C04488=1085.329,-36.806,-55.237,174.337,18.373,153.014
C04489=1085.323,-37.056,-55.224,174.335,18.371,153.014
C04490=1085.317,-37.305,-55.212,174.334,18.370,153.014
C04491=1085.311,-37.555,-55.200,174.332,18.367,153.013
C04492=1085.305,-37.805,-55.188,174.330,18.365,153.013
C04493=1085.300,-38.054,-55.175,174.329,18.364,153.013
C04494=1085.294,-38.304,-55.163,174.328,18.362,153.013
C04495=1085.288,-38.554,-55.150,174.326,18.361,153.013
C04496=1085.282,-38.802,-55.139,174.325,18.359,153.013
C04497=1085.276,-39.052,-55.126,174.323,18.358,153.013
C04498=1085.270,-39.302,-55.114,174.321,18.356,153.013
C04499=1085.264,-39.552,-55.102,174.320,18.353,153.013
C04500=1085.258,-39.802,-55.090,174.318,18.352,153.013
C04501=1085.252,-40.051,-55.078,174.317,18.350,153.013
C04502=1085.246,-40.301,-55.066,174.316,18.349,153.013
C04503=1085.240,-40.551,-55.053,174.314,18.347,153.013
C04504=1085.234,-40.800,-55.041,174.313,18.346,153.013
C04505=1085.228,-41.050,-55.029,174.311,18.344,153.013
C04506=1085.222,-41.300,-55.016,174.309,18.342,153.013
C04507=1085.217,-41.549,-55.004,174.308,18.341,153.013
C04508=1085.210,-41.798,-54.992,174.306,18.339,153.013
C04509=1085.204,-42.048,-54.980,174.305,18.337,153.013
C04510=1085.198,-42.299,-54.968,174.303,18.336,153.013
C04511=1085.192,-42.548,-54.956,174.302,18.334,153.013
C04512=1085.186,-42.797,-54.944,174.301,18.333,153.013
C04513=1085.181,-43.047,-54.931,174.299,18.331,153.013
C04514=1085.175,-43.296,-54.919,174.297,18.329,153.013
C04515=1085.169,-43.546,-54.907,174.296,18.328,153.013
C04516=1085.162,-43.796,-54.896,174.294,18.326,153.012
C04517=1085.157,-44.045,-54.884,174.293,18.324,153.012
C04518=1085.151,-44.295,-54.871,174.292,18.322,153.012
C04519=1085.144,-44.545,-54.859,174.290,18.321,153.012
C04520=1085.139,-44.794,-54.847,174.289,18.319,153.012
C04521=1085.133,-45.044,-54.834,174.287,18.318,153.012
C04522=1085.127,-45.293,-54.823,174.286,18.316,153.012
C04523=1085.122,-45.543,-54.811,174.284,18.314,153.012
C04524=1085.115,-45.793,-54.799,174.282,18.313,153.012
C04525=1085.110,-46.042,-54.787,174.281,18.311,153.012
C04526=1085.104,-46.293,-54.775,174.279,18.309,153.012
C04527=1085.097,-46.542,-54.763,174.278,18.308,153.012
C04528=1085.092,-46.791,-54.751,174.277,18.306,153.012
C04529=1085.085,-47.041,-54.739,174.275,18.305,153.012
C04530=1085.080,-47.291,-54.727,174.274,18.303,153.012
C04531=1085.074,-47.540,-54.715,174.272,18.302,153.012
C04532=1085.068,-47.790,-54.703,174.270,18.300,153.012
C04533=1085.063,-48.040,-54.691,174.269,18.298,153.012
C04534=1085.056,-48.290,-54.679,174.267,18.297,153.012
C04535=1085.051,-48.539,-54.667,174.266,18.295,153.012
C04536=1085.044,-48.812,-54.654,174.264,18.293,153.012
C04537=1085.038,-49.083,-54.641,174.263,18.292,153.012
C04538=1085.031,-49.356,-54.628,174.261,18.289,153.011
C04539=1085.025,-49.629,-54.615,174.260,18.288,153.011
C04540=1085.019,-49.878,-54.603,174.258,18.286,153.011
C04541=1085.013,-50.127,-54.591,174.257,18.285,153.011
C04542=1085.007,-50.378,-54.580,174.255,18.283,153.011
C04543=1085.002,-50.627,-54.568,174.254,18.282,153.011
C04544=1084.995,-50.876,-54.556,174.253,18.280,153.011
C04545=1084.989,-51.127,-54.545,174.251,18.279,153.011
C04546=1084.983,-51.376,-54.532,174.249,18.277,153.011
C04547=1084.977,-51.626,-54.521,174.247,18.275,153.011
C04548=1084.971,-51.875,-54.510,174.246,18.274,153.011
C04549=1084.965,-52.125,-54.497,174.244,18.272,153.011
C04550=1084.959,-52.375,-54.486,174.243,18.271,153.011
C04551=1084.953,-52.624,-54.474,174.242,18.269,153.011
C04552=1084.946,-52.874,-54.463,174.240,18.268,153.011
C04553=1084.941,-53.124,-54.450,174.238,18.266,153.011
C04554=1084.934,-53.373,-54.439,174.237,18.265,153.011
C04555=1084.928,-53.623,-54.428,174.236,18.263,153.011
C04556=1084.923,-53.872,-54.415,174.234,18.262,153.011
C04557=1084.916,-54.122,-54.404,174.233,18.260,153.011
C04558=1084.910,-54.372,-54.392,174.231,18.259,153.011
C04559=1084.904,-54.621,-54.381,174.229,18.257,153.011
C04560=1084.898,-54.871,-54.369,174.227,18.256,153.011
C04561=1084.892,-55.121,-54.358,174.226,18.254,153.011
C04562=1084.886,-55.370,-54.346,174.225,18.252,153.011
C04563=1084.881,-55.620,-54.334,174.223,18.251,153.011
C04564=1084.874,-55.870,-54.322,174.222,18.249,153.011
C04565=1084.868,-56.120,-54.311,174.220,18.248,153.011
C04566=1084.862,-56.369,-54.300,174.219,18.246,153.011
C04567=1084.856,-56.619,-54.288,174.217,18.245,153.011
C04568=1084.850,-56.868,-54.276,174.216,18.244,153.011
C04569=1084.844,-57.118,-54.265,174.215,18.242,153.011
C04570=1084.838,-57.367,-54.253,174.213,18.241,153.011
C04571=1084.832,-57.618,-54.242,174.212,18.239,153.011
C04572=1084.826,-57.866,-54.230,174.210,18.237,153.011
C04573=1084.820,-58.117,-54.219,174.209,18.236,153.011
C04574=1084.814,-58.366,-54.208,174.207,18.235,153.011
C04575=1084.808,-58.616,-54.195,174.206,18.233,153.011
C04576=1084.802,-58.866,-54.184,174.204,18.231,153.011
C04577=1084.796,-59.115,-54.172,174.202,18.230,153.011
C04578=1084.790,-59.365,-54.162,174.201,18.228,153.011
C04579=1084.784,-59.615,-54.150,174.199,18.227,153.011
C04580=1084.778,-59.864,-54.138,174.198,18.226,153.011
C04581=1084.772,-60.114,-54.127,174.196,18.224,153.011
C04582=1084.766,-60.363,-54.115,174.195,18.222,153.011
C04583=1084.760,-60.613,-54.104,174.193,18.221,153.011
C04584=1084.754,-60.863,-54.093,174.192,18.219,153.011
C04585=1084.748,-61.113,-54.081,174.190,18.218,153.011
C04586=1084.742,-61.362,-54.070,174.189,18.217,153.011
C04587=1084.736,-61.612,-54.058,174.187,18.215,153.011
C04588=1084.730,-61.861,-54.047,174.186,18.214,153.011
C04589=1084.723,-62.111,-54.036,174.185,18.212,153.011
C04590=1084.718,-62.361,-54.024,174.183,18.211,153.011
C04591=1084.712,-62.610,-54.013,174.182,18.209,153.011
C04592=1084.706,-62.860,-54.001,174.180,18.208,153.011
C04593=1084.700,-63.110,-53.990,174.179,18.206,153.011
C04594=1084.694,-63.359,-53.979,174.177,18.205,153.011
C04595=1084.689,-63.609,-53.967,174.176,18.204,153.011
C04596=1084.682,-63.859,-53.956,174.174,18.202,153.011
C04597=1084.677,-64.109,-53.945,174.173,18.201,153.011
C04598=1084.671,-64.358,-53.933,174.171,18.199,153.011
C04599=1084.664,-64.608,-53.922,174.170,18.198,153.011
C04600=1084.658,-64.881,-53.910,174.168,18.196,153.011
C04601=1084.652,-65.155,-53.898,174.166,18.194,153.011
C04602=1084.645,-65.429,-53.885,174.165,18.193,153.011
C04603=1084.638,-65.703,-53.873,174.163,18.191,153.011
C04604=1084.632,-65.952,-53.861,174.162,18.190,153.011
C04605=1084.627,-66.201,-53.850,174.160,18.188,153.011
C04606=1084.620,-66.451,-53.839,174.159,18.187,153.011
C04607=1084.615,-66.701,-53.828,174.157,18.186,153.011
C04608=1084.609,-66.951,-53.816,174.156,18.184,153.011
C04609=1084.603,-67.200,-53.805,174.155,18.182,153.011
C04610=1084.597,-67.450,-53.794,174.153,18.181,153.011
C04611=1084.591,-67.700,-53.783,174.151,18.179,153.011
C04612=1084.585,-67.950,-53.772,174.149,18.178,153.011
C04613=1084.579,-68.199,-53.761,174.148,18.176,153.011
C04614=1084.573,-68.449,-53.750,174.146,18.175,153.011
C04615=1084.567,-68.698,-53.738,174.145,18.174,153.011
C04616=1084.562,-68.948,-53.727,174.143,18.172,153.011
C04617=1084.556,-69.198,-53.715,174.142,18.171,153.011
C04618=1084.550,-69.448,-53.704,174.140,18.169,153.011
C04619=1084.544,-69.697,-53.694,174.139,18.168,153.011
C04620=1084.538,-69.947,-53.682,174.137,18.166,153.011
C04621=1084.532,-70.197,-53.671,174.136,18.165,153.011
C04622=1084.526,-70.446,-53.661,174.134,18.164,153.011
C04623=1084.520,-70.696,-53.649,174.133,18.162,153.011
C04624=1084.514,-70.945,-53.638,174.132,18.161,153.011
C04625=1084.508,-71.195,-53.627,174.130,18.160,153.011
C04626=1084.503,-71.445,-53.615,174.128,18.158,153.011
C04627=1084.497,-71.695,-53.604,174.127,18.156,153.011
C04628=1084.491,-71.944,-53.593,174.126,18.155,153.011
C04629=1084.485,-72.194,-53.582,174.124,18.154,153.011
C04630=1084.479,-72.444,-53.571,174.123,18.152,153.011
C04631=1084.473,-72.693,-53.560,174.121,18.151,153.011
C04632=1084.468,-72.943,-53.549,174.119,18.150,153.011
C04633=1084.461,-73.193,-53.538,174.118,18.148,153.011
C04634=1084.455,-73.443,-53.527,174.117,18.147,153.011
C04635=1084.450,-73.692,-53.516,174.115,18.146,153.011
C04636=1084.444,-73.942,-53.506,174.114,18.144,153.011
C04637=1084.438,-74.192,-53.494,174.112,18.142,153.011
C04638=1084.432,-74.441,-53.483,174.110,18.141,153.011
C04639=1084.426,-74.691,-53.473,174.109,18.140,153.011
C04640=1084.420,-74.941,-53.461,174.108,18.138,153.011
C04641=1084.414,-75.190,-53.450,174.107,18.138,153.011
C04642=1084.408,-75.440,-53.440,174.105,18.136,153.011
C04643=1084.401,-75.690,-53.429,174.104,18.135,153.011
C04644=1084.396,-75.939,-53.418,174.102,18.134,153.011
C04645=1084.390,-76.189,-53.407,174.101,18.133,153.011
C04646=1084.384,-76.438,-53.396,174.099,18.131,153.011
C04647=1084.378,-76.688,-53.385,174.098,18.129,153.011
C04648=1084.372,-76.938,-53.374,174.096,18.128,153.011
C04649=1084.366,-77.187,-53.363,174.095,18.127,153.011
C04650=1084.359,-77.437,-53.353,174.093,18.126,153.011
C04651=1084.354,-77.687,-53.342,174.092,18.124,153.011
C04652=1084.348,-77.937,-53.332,174.090,18.123,153.011
C04653=1084.342,-78.186,-53.321,174.089,18.122,153.011
C04654=1084.336,-78.437,-53.309,174.087,18.120,153.011
C04655=1084.330,-78.686,-53.299,174.086,18.119,153.011
C04656=1084.324,-78.935,-53.288,174.084,18.118,153.011
C04657=1084.318,-79.185,-53.277,174.082,18.117,153.011
C04658=1084.312,-79.435,-53.266,174.081,18.115,153.011
C04659=1084.306,-79.685,-53.256,174.079,18.114,153.012
C04660=1084.300,-79.935,-53.245,174.078,18.112,153.012
C04661=1084.294,-80.184,-53.235,174.076,18.111,153.012
C04662=1084.288,-80.434,-53.224,174.075,18.110,153.012
C04663=1084.282,-80.683,-53.213,174.073,18.109,153.012
C04664=1084.275,-80.960,-53.201,174.072,18.107,153.012
C04665=1084.268,-81.235,-53.189,174.070,18.106,153.012
C04666=1084.262,-81.511,-53.178,174.069,18.105,153.012
C04667=1084.254,-81.787,-53.166,174.067,18.104,153.012
C04668=1084.249,-82.037,-53.155,174.065,18.102,153.012
C04669=1084.242,-82.286,-53.145,174.064,18.101,153.012
C04670=1084.236,-82.536,-53.134,174.062,18.100,153.012
C04671=1084.230,-82.786,-53.123,174.061,18.098,153.012
C04672=1084.224,-83.035,-53.113,174.059,18.097,153.012
C04673=1084.218,-83.285,-53.103,174.058,18.096,153.012
C04674=1084.212,-83.535,-53.091,174.056,18.095,153.012
C04675=1084.206,-83.784,-53.081,174.054,18.094,153.012
C04676=1084.200,-84.034,-53.070,174.053,18.092,153.012
C04677=1084.194,-84.283,-53.061,174.051,18.091,153.012
C04678=1084.187,-84.534,-53.049,174.050,18.089,153.012
C04679=1084.182,-84.783,-53.038,174.048,18.088,153.012
C04680=1084.175,-85.033,-53.029,174.047,18.087,153.013
C04681=1084.170,-85.282,-53.018,174.046,18.086,153.013
C04682=1084.164,-85.532,-53.007,174.044,18.085,153.013
C04683=1084.157,-85.782,-52.997,174.043,18.084,153.013
C04684=1084.151,-86.032,-52.986,174.041,18.083,153.013
C04685=1084.145,-86.281,-52.976,174.040,18.082,153.013
C04686=1084.139,-86.531,-52.965,174.038,18.080,153.013
C04687=1084.134,-86.781,-52.955,174.037,18.079,153.013
C04688=1084.127,-87.031,-52.944,174.035,18.078,153.013
C04689=1084.121,-87.280,-52.934,174.033,18.077,153.013
C04690=1084.115,-87.530,-52.924,174.032,18.075,153.013
C04691=1084.109,-87.779,-52.913,174.030,18.074,153.013
C04692=1084.103,-88.029,-52.903,174.029,18.073,153.013
C04693=1084.097,-88.279,-52.892,174.028,18.072,153.013
C04694=1084.091,-88.529,-52.881,174.026,18.071,153.013
C04695=1084.084,-88.778,-52.871,174.025,18.070,153.013
C04696=1084.079,-89.028,-52.861,174.023,18.069,153.013
C04697=1084.072,-89.277,-52.851,174.021,18.068,153.014
C04698=1084.067,-89.527,-52.840,174.020,18.066,153.014
C04699=1084.060,-89.777,-52.830,174.018,18.065,153.014
C04700=1084.054,-90.027,-52.819,174.017,18.064,153.014
C04701=1084.049,-90.277,-52.809,174.015,18.062,153.014
C04702=1084.042,-90.526,-52.799,174.014,18.061,153.014
C04703=1084.037,-90.776,-52.788,174.012,18.060,153.014
C04704=1084.030,-91.025,-52.778,174.011,18.059,153.014
C04705=1084.025,-91.275,-52.768,174.010,18.058,153.014
C04706=1084.018,-91.525,-52.758,174.008,18.057,153.014
C04707=1084.012,-91.775,-52.746,174.007,18.056,153.014
C04708=1084.006,-92.025,-52.737,174.005,18.055,153.014
C04709=1084.000,-92.274,-52.726,174.003,18.054,153.014
C04710=1083.994,-92.524,-52.716,174.002,18.052,153.014
C04711=1083.988,-92.773,-52.705,174.000,18.051,153.014
C04712=1083.983,-93.024,-52.695,173.999,18.050,153.014
C04713=1083.976,-93.273,-52.685,173.997,18.049,153.015
C04714=1083.971,-93.523,-52.675,173.996,18.048,153.014
C04715=1083.964,-93.772,-52.665,173.995,18.047,153.015
C04716=1083.959,-94.022,-52.654,173.993,18.046,153.015
C04717=1083.952,-94.272,-52.644,173.991,18.045,153.015
C04718=1083.947,-94.522,-52.634,173.990,18.043,153.015
C04719=1083.940,-94.771,-52.623,173.988,18.042,153.015
C04720=1083.935,-95.021,-52.613,173.987,18.041,153.015
C04721=1083.928,-95.271,-52.603,173.985,18.040,153.015
C04722=1083.923,-95.521,-52.593,173.983,18.039,153.015
C04723=1083.917,-95.770,-52.583,173.983,18.038,153.015
C04724=1083.911,-96.020,-52.572,173.981,18.037,153.015
C04725=1083.905,-96.270,-52.563,173.979,18.036,153.015
C04726=1083.899,-96.519,-52.552,173.978,18.034,153.015
C04727=1083.893,-96.769,-52.542,173.976,18.033,153.015
C04728=1083.886,-97.047,-52.531,173.975,18.032,153.016
C04729=1083.879,-97.325,-52.520,173.973,18.031,153.016
C04730=1083.873,-97.603,-52.508,173.971,18.030,153.016
C04731=1083.866,-97.881,-52.497,173.970,18.029,153.016
C04732=1083.860,-98.131,-52.487,173.968,18.028,153.016
C04733=1083.854,-98.381,-52.477,173.966,18.027,153.016
C04734=1083.847,-98.631,-52.467,173.965,18.026,153.016
C04735=1083.842,-98.881,-52.457,173.963,18.025,153.016
C04736=1083.835,-99.130,-52.446,173.961,18.024,153.016
C04737=1083.829,-99.380,-52.437,173.961,18.022,153.016
C04738=1083.824,-99.630,-52.427,173.959,18.021,153.016
C04739=1083.817,-99.879,-52.416,173.958,18.020,153.016
C04740=1083.811,-100.129,-52.407,173.956,18.019,153.017
C04741=1083.805,-100.379,-52.397,173.954,18.018,153.017
C04742=1083.799,-100.628,-52.386,173.953,18.017,153.017
C04743=1083.793,-100.878,-52.377,173.951,18.016,153.017
C04744=1083.787,-101.128,-52.367,173.950,18.016,153.017
C04745=1083.781,-101.377,-52.356,173.948,18.015,153.017
C04746=1083.775,-101.627,-52.347,173.947,18.014,153.017
C04747=1083.769,-101.877,-52.337,173.945,18.013,153.017
C04748=1083.762,-102.127,-52.328,173.944,18.011,153.017
C04749=1083.757,-102.376,-52.317,173.942,18.010,153.017
C04750=1083.751,-102.626,-52.307,173.941,18.009,153.018
C04751=1083.744,-102.876,-52.298,173.939,18.008,153.018
C04752=1083.738,-103.125,-52.287,173.938,18.007,153.018
C04753=1083.732,-103.375,-52.277,173.936,18.006,153.018
C04754=1083.726,-103.625,-52.267,173.934,18.005,153.018
C04755=1083.719,-103.875,-52.258,173.933,18.004,153.018
C04756=1083.713,-104.124,-52.247,173.932,18.004,153.018
C04757=1083.708,-104.375,-52.237,173.930,18.003,153.018
C04758=1083.701,-104.624,-52.228,173.929,18.002,153.018
C04759=1083.695,-104.874,-52.218,173.927,18.001,153.018
C04760=1083.690,-105.123,-52.209,173.925,18.000,153.019
C04761=1083.684,-105.373,-52.198,173.924,17.999,153.019
C04762=1083.678,-105.622,-52.188,173.923,17.998,153.019
C04763=1083.672,-105.872,-52.179,173.921,17.997,153.019
C04764=1083.665,-106.122,-52.169,173.919,17.996,153.019
C04765=1083.659,-106.372,-52.160,173.918,17.995,153.019
C04766=1083.653,-106.621,-52.149,173.916,17.994,153.019
C04767=1083.647,-106.871,-52.139,173.914,17.993,153.019
C04768=1083.641,-107.121,-52.130,173.914,17.992,153.019
C04769=1083.635,-107.371,-52.120,173.912,17.991,153.020
C04770=1083.629,-107.621,-52.111,173.910,17.990,153.020
C04771=1083.623,-107.870,-52.101,173.909,17.989,153.020
C04772=1083.617,-108.120,-52.090,173.907,17.988,153.020
C04773=1083.611,-108.370,-52.081,173.906,17.988,153.020
C04774=1083.605,-108.619,-52.071,173.904,17.987,153.020
C04775=1083.598,-108.869,-52.061,173.903,17.986,153.020
C04776=1083.592,-109.119,-52.052,173.901,17.985,153.020
C04777=1083.586,-109.369,-52.042,173.899,17.984,153.021
C04778=1083.580,-109.619,-52.033,173.898,17.984,153.021
C04779=1083.574,-109.868,-52.023,173.897,17.983,153.021
C04780=1083.567,-110.118,-52.013,173.895,17.981,153.021
C04781=1083.561,-110.367,-52.003,173.893,17.980,153.021
C04782=1083.555,-110.617,-51.994,173.892,17.979,153.021
C04783=1083.549,-110.867,-51.984,173.891,17.979,153.021
C04784=1083.543,-111.117,-51.974,173.889,17.978,153.021
C04785=1083.537,-111.367,-51.964,173.887,17.977,153.022
C04786=1083.531,-111.617,-51.955,173.885,17.976,153.022
C04787=1083.525,-111.867,-51.945,173.884,17.975,153.022
C04788=1083.519,-112.116,-51.936,173.883,17.975,153.022
C04789=1083.513,-112.365,-51.926,173.881,17.974,153.022
C04790=1083.507,-112.615,-51.917,173.880,17.973,153.022
C04791=1083.501,-112.865,-51.907,173.878,17.972,153.022
C04792=1083.494,-113.139,-51.896,173.876,17.971,153.022
C04793=1083.487,-113.413,-51.886,173.874,17.970,153.023
C04794=1083.481,-113.687,-51.875,173.873,17.969,153.023
C04795=1083.474,-113.962,-51.866,173.871,17.968,153.023
C04796=1083.467,-114.211,-51.856,173.870,17.967,153.023
C04797=1083.462,-114.462,-51.846,173.868,17.967,153.023
C04798=1083.455,-114.711,-51.837,173.867,17.966,153.023
C04799=1083.449,-114.961,-51.827,173.865,17.965,153.023
C04800=1083.443,-115.211,-51.818,173.863,17.964,153.023
C04801=1083.437,-115.460,-51.808,173.862,17.963,153.024
C04802=1083.430,-115.710,-51.799,173.860,17.963,153.024
C04803=1083.425,-115.959,-51.790,173.859,17.962,153.024
C04804=1083.419,-116.209,-51.780,173.857,17.961,153.024
C04805=1083.412,-116.459,-51.770,173.856,17.960,153.024
C04806=1083.406,-116.709,-51.761,173.854,17.960,153.024
C04807=1083.400,-116.958,-51.751,173.853,17.959,153.024
C04808=1083.394,-117.208,-51.742,173.851,17.958,153.025
C04809=1083.388,-117.458,-51.732,173.850,17.957,153.025
C04810=1083.382,-117.708,-51.723,173.848,17.957,153.025
C04811=1083.375,-117.958,-51.713,173.847,17.956,153.025
C04812=1083.370,-118.207,-51.705,173.845,17.955,153.025
C04813=1083.364,-118.457,-51.695,173.844,17.955,153.025
C04814=1083.357,-118.707,-51.686,173.842,17.954,153.025
C04815=1083.351,-118.956,-51.676,173.840,17.952,153.026
C04816=1083.345,-119.206,-51.667,173.839,17.952,153.026
C04817=1083.339,-119.456,-51.657,173.838,17.951,153.026
C04818=1083.332,-119.706,-51.648,173.836,17.950,153.026
C04819=1083.326,-119.956,-51.638,173.834,17.950,153.026
C04820=1083.321,-120.205,-51.630,173.832,17.949,153.026
C04821=1083.315,-120.455,-51.620,173.832,17.948,153.026
C04822=1083.309,-120.705,-51.611,173.830,17.948,153.027
C04823=1083.302,-120.954,-51.602,173.828,17.947,153.027
C04824=1083.296,-121.204,-51.592,173.826,17.946,153.027
C04825=1083.289,-121.454,-51.582,173.825,17.946,153.027
C04826=1083.284,-121.704,-51.574,173.824,17.945,153.027
C04827=1083.278,-121.954,-51.564,173.822,17.944,153.027
C04828=1083.272,-122.203,-51.555,173.820,17.943,153.028
C04829=1083.265,-122.453,-51.546,173.819,17.943,153.028
C04830=1083.259,-122.703,-51.536,173.817,17.942,153.028
C04831=1083.253,-122.953,-51.527,173.815,17.941,153.028
C04832=1083.247,-123.202,-51.518,173.814,17.940,153.028
C04833=1083.241,-123.452,-51.509,173.813,17.940,153.028
C04834=1083.235,-123.702,-51.499,173.811,17.939,153.029
C04835=1083.228,-123.952,-51.491,173.809,17.938,153.029
C04836=1083.222,-124.202,-51.481,173.807,17.938,153.029
C04837=1083.217,-124.451,-51.472,173.807,17.937,153.029
C04838=1083.210,-124.701,-51.463,173.805,17.936,153.029
C04839=1083.205,-124.951,-51.454,173.803,17.935,153.029
C04840=1083.198,-125.200,-51.445,173.802,17.935,153.030
C04841=1083.191,-125.450,-51.435,173.800,17.934,153.030
C04842=1083.185,-125.700,-51.426,173.799,17.933,153.030
C04843=1083.179,-125.949,-51.418,173.797,17.933,153.030
C04844=1083.173,-126.199,-51.408,173.796,17.932,153.030
C04845=1083.167,-126.449,-51.399,173.794,17.932,153.030
C04846=1083.161,-126.699,-51.390,173.792,17.931,153.031
C04847=1083.154,-126.949,-51.381,173.791,17.931,153.031
C04848=1083.149,-127.198,-51.372,173.789,17.930,153.031
C04849=1083.142,-127.448,-51.362,173.787,17.929,153.031
C04850=1083.136,-127.698,-51.354,173.786,17.928,153.031
C04851=1083.130,-127.948,-51.344,173.785,17.928,153.031
C04852=1083.125,-128.205,-51.335,173.783,17.927,153.032
C04853=1083.124,-128.460,-51.324,173.782,17.925,153.031
C04854=1083.128,-128.715,-51.311,173.782,17.921,153.031
C04855=1083.136,-128.967,-51.297,173.782,17.917,153.030
C04856=1082.735,-128.989,-51.433,173.737,18.034,153.060
C04857=1082.727,-128.736,-51.447,173.738,18.039,153.061
C04858=1082.724,-128.481,-51.459,173.739,18.042,153.061
C04859=1082.724,-128.226,-51.470,173.740,18.044,153.062
C04860=1082.728,-127.970,-51.481,173.740,18.045,153.062
C04861=1082.735,-127.720,-51.490,173.742,18.046,153.061
C04862=1082.740,-127.471,-51.498,173.744,18.047,153.061
C04863=1082.747,-127.221,-51.508,173.746,18.047,153.061
C04864=1082.754,-126.971,-51.517,173.747,18.048,153.061
C04865=1082.759,-126.721,-51.526,173.749,18.048,153.061
C04866=1082.766,-126.471,-51.535,173.750,18.050,153.061
C04867=1082.771,-126.222,-51.544,173.751,18.049,153.060
C04868=1082.778,-125.972,-51.553,173.753,18.051,153.060
C04869=1082.784,-125.722,-51.562,173.755,18.051,153.060
C04870=1082.790,-125.472,-51.572,173.757,18.052,153.060
C04871=1082.797,-125.223,-51.581,173.757,18.053,153.060
C04872=1082.803,-124.972,-51.590,173.759,18.053,153.060
C04873=1082.808,-124.723,-51.599,173.761,18.054,153.059
C04874=1082.815,-124.473,-51.608,173.762,18.054,153.059
C04875=1082.822,-124.224,-51.617,173.764,18.055,153.059
C04876=1082.827,-123.974,-51.626,173.766,18.056,153.059
C04877=1082.834,-123.724,-51.636,173.767,18.057,153.059
C04878=1082.839,-123.475,-51.645,173.768,18.057,153.059
C04879=1082.845,-123.225,-51.654,173.770,18.058,153.058
C04880=1082.851,-122.974,-51.663,173.772,18.059,153.058
C04881=1082.858,-122.725,-51.672,173.774,18.060,153.058
C04882=1082.864,-122.475,-51.682,173.775,18.060,153.058
C04883=1082.870,-122.226,-51.691,173.776,18.061,153.058
C04884=1082.876,-121.976,-51.701,173.778,18.062,153.058
C04885=1082.882,-121.726,-51.709,173.780,18.062,153.058
C04886=1082.888,-121.476,-51.719,173.781,18.063,153.057
C04887=1082.895,-121.227,-51.728,173.782,18.064,153.057
C04888=1082.901,-120.977,-51.738,173.784,18.064,153.057
C04889=1082.907,-120.727,-51.747,173.786,18.065,153.057
C04890=1082.913,-120.477,-51.756,173.787,18.066,153.057
C04891=1082.919,-120.227,-51.765,173.789,18.066,153.057
C04892=1082.925,-119.978,-51.775,173.791,18.067,153.057
C04893=1082.931,-119.728,-51.784,173.792,18.068,153.056
C04894=1082.937,-119.478,-51.794,173.793,18.069,153.056
C04895=1082.944,-119.229,-51.803,173.795,18.069,153.056
C04896=1082.950,-118.979,-51.812,173.797,18.070,153.056
C04897=1082.956,-118.730,-51.822,173.798,18.072,153.056
C04898=1082.962,-118.479,-51.830,173.799,18.072,153.056
C04899=1082.968,-118.229,-51.840,173.801,18.073,153.055
C04900=1082.974,-117.980,-51.850,173.803,18.074,153.055
C04901=1082.980,-117.730,-51.859,173.804,18.075,153.055
C04902=1082.986,-117.480,-51.869,173.806,18.075,153.055
C04903=1082.993,-117.230,-51.878,173.807,18.076,153.055
C04904=1082.999,-116.980,-51.888,173.809,18.077,153.055
C04905=1083.004,-116.731,-51.897,173.811,18.078,153.055
C04906=1083.011,-116.482,-51.907,173.813,18.078,153.054
C04907=1083.017,-116.232,-51.916,173.813,18.079,153.054
C04908=1083.024,-115.982,-51.925,173.815,18.080,153.054
C04909=1083.030,-115.732,-51.935,173.817,18.081,153.054
C04910=1083.036,-115.483,-51.944,173.818,18.082,153.054
C04911=1083.042,-115.232,-51.953,173.819,18.082,153.054
C04912=1083.048,-114.982,-51.963,173.821,18.083,153.054
C04913=1083.054,-114.733,-51.972,173.823,18.084,153.054
C04914=1083.060,-114.483,-51.982,173.824,18.085,153.053
C04915=1083.066,-114.234,-51.991,173.826,18.086,153.053
C04916=1083.072,-113.984,-52.001,173.827,18.086,153.053
C04917=1083.079,-113.709,-52.012,173.829,18.087,153.053
C04918=1083.086,-113.435,-52.022,173.831,18.088,153.053
C04919=1083.093,-113.161,-52.033,173.832,18.089,153.053
C04920=1083.099,-112.886,-52.043,173.834,18.090,153.053
C04921=1083.105,-112.637,-52.053,173.836,18.091,153.053
C04922=1083.111,-112.387,-52.062,173.837,18.092,153.052
C04923=1083.118,-112.137,-52.072,173.839,18.093,153.052
C04924=1083.124,-111.887,-52.082,173.840,18.093,153.052
C04925=1083.130,-111.637,-52.091,173.842,18.094,153.052
C04926=1083.136,-111.388,-52.101,173.843,18.095,153.052
C04927=1083.142,-111.138,-52.110,173.845,18.096,153.052
C04928=1083.148,-110.888,-52.120,173.847,18.097,153.052
C04929=1083.154,-110.638,-52.130,173.848,18.098,153.052
C04930=1083.159,-110.389,-52.139,173.849,18.099,153.051
C04931=1083.166,-110.140,-52.149,173.851,18.100,153.051
C04932=1083.172,-109.890,-52.159,173.853,18.101,153.051
C04933=1083.178,-109.640,-52.169,173.854,18.102,153.051
C04934=1083.184,-109.390,-52.178,173.855,18.102,153.051
C04935=1083.191,-109.140,-52.188,173.857,18.103,153.051
C04936=1083.197,-108.891,-52.197,173.859,18.104,153.051
C04937=1083.203,-108.641,-52.207,173.860,18.105,153.051
C04938=1083.209,-108.391,-52.216,173.862,18.106,153.050
C04939=1083.215,-108.141,-52.226,173.864,18.107,153.050
C04940=1083.221,-107.892,-52.237,173.865,18.108,153.050
C04941=1083.227,-107.642,-52.246,173.866,18.109,153.050
C04942=1083.233,-107.392,-52.256,173.868,18.110,153.050
C04943=1083.239,-107.142,-52.266,173.870,18.111,153.050
C04944=1083.246,-106.892,-52.275,173.871,18.112,153.050
C04945=1083.252,-106.643,-52.285,173.872,18.112,153.050
C04946=1083.258,-106.393,-52.296,173.874,18.113,153.050
C04947=1083.264,-106.143,-52.305,173.875,18.114,153.050
C04948=1083.270,-105.894,-52.315,173.877,18.115,153.049
C04949=1083.276,-105.644,-52.324,173.879,18.116,153.049
C04950=1083.282,-105.394,-52.334,173.881,18.117,153.049
C04951=1083.288,-105.145,-52.345,173.881,18.118,153.049
C04952=1083.294,-104.895,-52.354,173.883,18.119,153.049
C04953=1083.300,-104.645,-52.364,173.885,18.120,153.049
C04954=1083.307,-104.395,-52.373,173.886,18.121,153.049
C04955=1083.312,-104.145,-52.384,173.888,18.123,153.049
C04956=1083.318,-103.896,-52.394,173.889,18.124,153.049
C04957=1083.325,-103.646,-52.403,173.890,18.124,153.049
C04958=1083.331,-103.396,-52.413,173.892,18.125,153.049
C04959=1083.336,-103.146,-52.423,173.894,18.126,153.048
C04960=1083.343,-102.897,-52.433,173.895,18.127,153.048
C04961=1083.349,-102.647,-52.443,173.897,18.128,153.048
C04962=1083.355,-102.397,-52.453,173.899,18.129,153.048
C04963=1083.361,-102.148,-52.463,173.900,18.130,153.048
C04964=1083.367,-101.898,-52.473,173.901,18.131,153.048
C04965=1083.373,-101.648,-52.483,173.903,18.132,153.048
C04966=1083.379,-101.398,-52.492,173.904,18.133,153.048
C04967=1083.385,-101.149,-52.503,173.906,18.134,153.048
C04968=1083.391,-100.899,-52.513,173.908,18.135,153.048
C04969=1083.397,-100.649,-52.522,173.909,18.136,153.047
C04970=1083.403,-100.400,-52.533,173.911,18.137,153.047
C04971=1083.409,-100.150,-52.543,173.912,18.138,153.047
C04972=1083.415,-99.900,-52.552,173.913,18.139,153.047
C04973=1083.423,-99.650,-52.563,173.915,18.140,153.047
C04974=1083.428,-99.400,-52.573,173.917,18.142,153.047
C04975=1083.434,-99.151,-52.583,173.918,18.143,153.047
C04976=1083.441,-98.901,-52.593,173.920,18.144,153.047
C04977=1083.446,-98.651,-52.603,173.922,18.145,153.047
C04978=1083.453,-98.402,-52.613,173.922,18.145,153.047
C04979=1083.459,-98.152,-52.623,173.924,18.146,153.047
C04980=1083.464,-97.902,-52.633,173.925,18.148,153.047
C04981=1083.471,-97.625,-52.644,173.927,18.149,153.046
C04982=1083.478,-97.347,-52.656,173.929,18.150,153.046
C04983=1083.485,-97.068,-52.667,173.931,18.151,153.046
C04984=1083.492,-96.790,-52.679,173.932,18.152,153.046
C04985=1083.497,-96.540,-52.689,173.934,18.153,153.046
C04986=1083.503,-96.290,-52.698,173.935,18.155,153.046
C04987=1083.509,-96.040,-52.709,173.937,18.156,153.046
C04988=1083.515,-95.790,-52.719,173.938,18.157,153.046
C04989=1083.521,-95.541,-52.730,173.940,18.158,153.046
C04990=1083.527,-95.291,-52.739,173.942,18.159,153.046
C04991=1083.533,-95.042,-52.750,173.943,18.161,153.046
C04992=1083.539,-94.792,-52.760,173.945,18.162,153.046
C04993=1083.545,-94.542,-52.770,173.946,18.162,153.046
C04994=1083.551,-94.293,-52.780,173.947,18.163,153.045
C04995=1083.557,-94.043,-52.791,173.949,18.165,153.045
C04996=1083.563,-93.793,-52.800,173.950,18.166,153.045
C04997=1083.569,-93.543,-52.812,173.952,18.167,153.045
C04998=1083.575,-93.293,-52.821,173.953,18.168,153.045
C04999=1083.581,-93.044,-52.832,173.955,18.170,153.045
C05000=1083.587,-92.794,-52.842,173.957,18.171,153.045
C05001=1083.593,-92.545,-52.853,173.958,18.172,153.045
C05002=1083.599,-92.295,-52.862,173.960,18.173,153.045
C05003=1083.605,-92.045,-52.873,173.961,18.174,153.045
C05004=1083.611,-91.795,-52.883,173.962,18.175,153.045
C05005=1083.617,-91.546,-52.893,173.964,18.176,153.045
C05006=1083.624,-91.295,-52.903,173.966,18.177,153.045
C05007=1083.629,-91.046,-52.914,173.967,18.179,153.045
C05008=1083.635,-90.796,-52.924,173.969,18.180,153.045
C05009=1083.641,-90.547,-52.935,173.970,18.181,153.045
C05010=1083.647,-90.297,-52.946,173.972,18.182,153.045
C05011=1083.653,-90.047,-52.955,173.973,18.183,153.044
C05012=1083.659,-89.798,-52.966,173.975,18.185,153.044
C05013=1083.666,-89.547,-52.976,173.976,18.186,153.044
C05014=1083.671,-89.298,-52.987,173.977,18.187,153.044
C05015=1083.678,-89.049,-52.997,173.979,18.188,153.044
C05016=1083.683,-88.799,-53.007,173.980,18.189,153.044
C05017=1083.689,-88.549,-53.018,173.982,18.190,153.044
C05018=1083.695,-88.300,-53.028,173.983,18.192,153.044
C05019=1083.702,-88.049,-53.039,173.985,18.193,153.044
C05020=1083.708,-87.800,-53.049,173.987,18.194,153.044
C05021=1083.713,-87.550,-53.059,173.988,18.195,153.044
C05022=1083.719,-87.300,-53.070,173.990,18.196,153.044
C05023=1083.726,-87.051,-53.081,173.991,18.198,153.044
C05024=1083.731,-86.801,-53.091,173.993,18.199,153.044
C05025=1083.738,-86.551,-53.101,173.994,18.201,153.044
C05026=1083.744,-86.302,-53.112,173.995,18.201,153.044
C05027=1083.750,-86.053,-53.123,173.997,18.202,153.044
C05028=1083.756,-85.802,-53.133,173.998,18.204,153.044
C05029=1083.762,-85.553,-53.144,174.000,18.205,153.044
C05030=1083.769,-85.303,-53.154,174.001,18.206,153.044
C05031=1083.774,-85.053,-53.164,174.003,18.207,153.043
C05032=1083.780,-84.803,-53.175,174.005,18.208,153.043
C05033=1083.786,-84.554,-53.186,174.006,18.210,153.043
C05034=1083.793,-84.304,-53.197,174.008,18.211,153.043
C05035=1083.799,-84.054,-53.206,174.009,18.212,153.043
C05036=1083.805,-83.805,-53.217,174.011,18.213,153.043
C05037=1083.810,-83.555,-53.228,174.012,18.215,153.043
C05038=1083.817,-83.305,-53.239,174.014,18.216,153.043
C05039=1083.823,-83.055,-53.249,174.015,18.218,153.043
C05040=1083.829,-82.806,-53.260,174.017,18.219,153.043
C05041=1083.835,-82.557,-53.270,174.019,18.220,153.043
C05042=1083.841,-82.306,-53.281,174.019,18.221,153.043
C05043=1083.847,-82.057,-53.292,174.021,18.222,153.043
C05044=1083.853,-81.807,-53.302,174.022,18.223,153.043
C05045=1083.860,-81.532,-53.314,174.024,18.224,153.043
C05046=1083.867,-81.255,-53.326,174.026,18.226,153.043
C05047=1083.873,-80.979,-53.338,174.028,18.227,153.043
C05048=1083.880,-80.704,-53.350,174.029,18.229,153.043
C05049=1083.887,-80.454,-53.360,174.031,18.230,153.043
C05050=1083.893,-80.204,-53.370,174.033,18.232,153.043
C05051=1083.898,-79.954,-53.381,174.034,18.233,153.043
C05052=1083.904,-79.705,-53.392,174.036,18.234,153.043
C05053=1083.911,-79.455,-53.403,174.037,18.236,153.043
C05054=1083.917,-79.205,-53.414,174.039,18.237,153.042
C05055=1083.923,-78.956,-53.425,174.040,18.238,153.043
C05056=1083.928,-78.706,-53.435,174.042,18.239,153.042
C05057=1083.935,-78.456,-53.447,174.043,18.241,153.042
C05058=1083.940,-78.206,-53.457,174.045,18.242,153.042
C05059=1083.947,-77.957,-53.467,174.046,18.243,153.042
C05060=1083.953,-77.707,-53.478,174.048,18.245,153.042
C05061=1083.959,-77.457,-53.489,174.049,18.246,153.042
C05062=1083.964,-77.208,-53.500,174.050,18.247,153.042
C05063=1083.970,-76.958,-53.511,174.052,18.248,153.042
C05064=1083.977,-76.708,-53.522,174.053,18.250,153.042
C05065=1083.983,-76.459,-53.533,174.055,18.251,153.042
C05066=1083.989,-76.209,-53.543,174.056,18.252,153.042
C05067=1083.995,-75.959,-53.555,174.058,18.254,153.042
C05068=1084.001,-75.710,-53.566,174.059,18.255,153.042
C05069=1084.007,-75.460,-53.576,174.061,18.256,153.042
C05070=1084.012,-75.211,-53.587,174.062,18.258,153.042
C05071=1084.019,-74.961,-53.599,174.064,18.259,153.042
C05072=1084.024,-74.711,-53.609,174.065,18.261,153.042
C05073=1084.031,-74.462,-53.620,174.067,18.262,153.042
C05074=1084.037,-74.212,-53.631,174.068,18.263,153.042
C05075=1084.043,-73.962,-53.642,174.070,18.265,153.042
C05076=1084.049,-73.713,-53.653,174.071,18.266,153.042
C05077=1084.055,-73.462,-53.664,174.073,18.268,153.042
C05078=1084.061,-73.213,-53.675,174.074,18.269,153.042
C05079=1084.066,-72.963,-53.686,174.076,18.270,153.042
C05080=1084.071,-72.714,-53.697,174.077,18.272,153.042
C05081=1084.078,-72.464,-53.708,174.079,18.273,153.042
C05082=1084.084,-72.214,-53.719,174.080,18.274,153.042
C05083=1084.089,-71.965,-53.730,174.082,18.276,153.042
C05084=1084.096,-71.714,-53.741,174.083,18.278,153.042
C05085=1084.101,-71.465,-53.752,174.084,18.279,153.042
C05086=1084.107,-71.215,-53.763,174.086,18.280,153.042
C05087=1084.113,-70.966,-53.774,174.087,18.282,153.042
C05088=1084.119,-70.716,-53.785,174.089,18.283,153.042
C05089=1084.125,-70.466,-53.796,174.090,18.285,153.042
C05090=1084.131,-70.217,-53.807,174.092,18.286,153.042
C05091=1084.137,-69.967,-53.818,174.093,18.287,153.042
C05092=1084.142,-69.717,-53.830,174.095,18.289,153.042
C05093=1084.148,-69.468,-53.841,174.096,18.291,153.042
C05094=1084.154,-69.218,-53.853,174.098,18.292,153.042
C05095=1084.160,-68.968,-53.863,174.099,18.293,153.042
C05096=1084.166,-68.719,-53.874,174.101,18.295,153.042
C05097=1084.172,-68.468,-53.886,174.102,18.296,153.042
C05098=1084.178,-68.219,-53.896,174.104,18.298,153.042
C05099=1084.184,-67.970,-53.908,174.105,18.299,153.042
C05100=1084.190,-67.720,-53.919,174.107,18.300,153.042
C05101=1084.195,-67.470,-53.931,174.108,18.302,153.042
C05102=1084.201,-67.221,-53.942,174.109,18.303,153.042
C05103=1084.207,-66.970,-53.953,174.111,18.305,153.042
C05104=1084.213,-66.721,-53.964,174.113,18.306,153.042
C05105=1084.220,-66.471,-53.976,174.114,18.308,153.042
C05106=1084.226,-66.222,-53.987,174.116,18.310,153.042
C05107=1084.231,-65.972,-53.997,174.118,18.311,153.042
C05108=1084.237,-65.722,-54.009,174.119,18.313,153.042
C05109=1084.243,-65.448,-54.022,174.121,18.314,153.042
C05110=1084.250,-65.175,-54.034,174.122,18.316,153.042
C05111=1084.257,-64.901,-54.046,174.124,18.317,153.042
C05112=1084.264,-64.628,-54.059,174.125,18.318,153.042
C05113=1084.269,-64.378,-54.070,174.127,18.321,153.042
C05114=1084.275,-64.128,-54.081,174.129,18.322,153.042
C05115=1084.281,-63.878,-54.092,174.130,18.324,153.042
C05116=1084.287,-63.629,-54.104,174.132,18.325,153.042
C05117=1084.293,-63.379,-54.115,174.133,18.327,153.042
C05118=1084.300,-63.129,-54.126,174.135,18.328,153.042
C05119=1084.305,-62.880,-54.139,174.136,18.329,153.042
C05120=1084.311,-62.630,-54.149,174.137,18.331,153.042
C05121=1084.317,-62.380,-54.161,174.139,18.332,153.042
C05122=1084.323,-62.131,-54.172,174.140,18.334,153.042
C05123=1084.329,-61.881,-54.184,174.142,18.336,153.042
C05124=1084.334,-61.631,-54.195,174.143,18.337,153.042
C05125=1084.341,-61.382,-54.207,174.145,18.338,153.042
C05126=1084.347,-61.132,-54.218,174.146,18.340,153.042
C05127=1084.353,-60.882,-54.229,174.148,18.341,153.042
C05128=1084.359,-60.633,-54.241,174.149,18.343,153.042
C05129=1084.365,-60.383,-54.252,174.150,18.344,153.042
C05130=1084.370,-60.133,-54.263,174.152,18.346,153.042
C05131=1084.377,-59.884,-54.275,174.154,18.347,153.042
C05132=1084.383,-59.634,-54.286,174.155,18.348,153.042
C05133=1084.389,-59.384,-54.297,174.156,18.350,153.042
C05134=1084.394,-59.135,-54.310,174.158,18.352,153.042
C05135=1084.401,-58.884,-54.321,174.159,18.353,153.042
C05136=1084.407,-58.636,-54.332,174.161,18.355,153.042
C05137=1084.413,-58.385,-54.344,174.163,18.357,153.043
C05138=1084.419,-58.136,-54.356,174.164,18.358,153.043
C05139=1084.425,-57.886,-54.367,174.166,18.360,153.043
C05140=1084.431,-57.637,-54.378,174.167,18.361,153.042
C05141=1084.437,-57.387,-54.390,174.169,18.362,153.043
C05142=1084.442,-57.137,-54.401,174.170,18.364,153.043
C05143=1084.449,-56.888,-54.413,174.172,18.365,153.043
C05144=1084.455,-56.638,-54.424,174.173,18.367,153.043
C05145=1084.461,-56.389,-54.436,174.175,18.369,153.043
C05146=1084.466,-56.139,-54.448,174.176,18.370,153.043
C05147=1084.473,-55.889,-54.460,174.177,18.372,153.043
C05148=1084.479,-55.639,-54.471,174.179,18.373,153.043
C05149=1084.485,-55.390,-54.483,174.180,18.374,153.043
C05150=1084.491,-55.140,-54.494,174.182,18.376,153.043
C05151=1084.497,-54.891,-54.506,174.183,18.377,153.043
C05152=1084.503,-54.641,-54.517,174.186,18.379,153.043
C05153=1084.509,-54.391,-54.529,174.187,18.381,153.043
C05154=1084.515,-54.141,-54.541,174.188,18.383,153.043
C05155=1084.522,-53.892,-54.553,174.190,18.384,153.043
C05156=1084.528,-53.643,-54.564,174.191,18.386,153.043
C05157=1084.533,-53.392,-54.576,174.193,18.387,153.043
C05158=1084.539,-53.143,-54.588,174.194,18.389,153.043
C05159=1084.546,-52.893,-54.599,174.195,18.390,153.043
C05160=1084.552,-52.643,-54.611,174.197,18.392,153.043
C05161=1084.557,-52.394,-54.622,174.199,18.393,153.043
C05162=1084.564,-52.144,-54.634,174.200,18.394,153.043
C05163=1084.570,-51.895,-54.646,174.201,18.396,153.043
C05164=1084.576,-51.645,-54.658,174.203,18.398,153.043
C05165=1084.582,-51.395,-54.670,174.205,18.400,153.043
C05166=1084.588,-51.146,-54.681,174.207,18.401,153.043
C05167=1084.594,-50.896,-54.693,174.208,18.403,153.043
C05168=1084.601,-50.646,-54.705,174.209,18.404,153.043
C05169=1084.606,-50.397,-54.716,174.211,18.406,153.043
C05170=1084.612,-50.147,-54.728,174.212,18.407,153.043
C05171=1084.617,-49.898,-54.741,174.214,18.409,153.043
C05172=1084.624,-49.648,-54.752,174.215,18.410,153.043
C05173=1084.631,-49.375,-54.766,174.216,18.412,153.043
C05174=1084.637,-49.103,-54.778,174.218,18.415,153.043
C05175=1084.643,-48.830,-54.791,174.220,18.416,153.043
C05176=1084.650,-48.558,-54.804,174.221,18.418,153.043
C05177=1084.655,-48.308,-54.816,174.223,18.419,153.044
C05178=1084.661,-48.059,-54.828,174.224,18.421,153.044
C05179=1084.667,-47.809,-54.840,174.226,18.423,153.044
C05180=1084.673,-47.560,-54.851,174.228,18.424,153.044
C05181=1084.679,-47.310,-54.864,174.229,18.426,153.044
C05182=1084.685,-47.060,-54.876,174.231,18.427,153.044
C05183=1084.691,-46.811,-54.888,174.232,18.429,153.044
C05184=1084.696,-46.560,-54.900,174.233,18.431,153.044
C05185=1084.703,-46.311,-54.912,174.235,18.433,153.044
C05186=1084.708,-46.062,-54.924,174.236,18.434,153.044
C05187=1084.714,-45.812,-54.936,174.237,18.436,153.044
C05188=1084.720,-45.562,-54.947,174.240,18.438,153.044
C05189=1084.726,-45.312,-54.960,174.241,18.439,153.044
C05190=1084.733,-45.063,-54.972,174.243,18.441,153.044
C05191=1084.738,-44.814,-54.984,174.244,18.442,153.044
C05192=1084.744,-44.564,-54.997,174.245,18.444,153.044
C05193=1084.750,-44.314,-55.008,174.247,18.446,153.044
C05194=1084.755,-44.064,-55.020,174.248,18.447,153.044
C05195=1084.762,-43.815,-55.032,174.249,18.449,153.044
C05196=1084.768,-43.565,-55.045,174.251,18.451,153.044
C05197=1084.773,-43.316,-55.057,174.253,18.453,153.044
C05198=1084.780,-43.066,-55.068,174.255,18.454,153.044
C05199=1084.786,-42.816,-55.080,174.256,18.456,153.044
C05200=1084.791,-42.567,-55.093,174.257,18.457,153.045
C05201=1084.798,-42.317,-55.105,174.259,18.459,153.045
C05202=1084.803,-42.067,-55.117,174.260,18.460,153.045
C05203=1084.809,-41.818,-55.129,174.262,18.462,153.045
C05204=1084.815,-41.568,-55.141,174.263,18.464,153.045
C05205=1084.821,-41.318,-55.154,174.265,18.466,153.045
C05206=1084.826,-41.069,-55.165,174.267,18.468,153.045
C05207=1084.833,-40.819,-55.177,174.268,18.469,153.045
C05208=1084.839,-40.569,-55.190,174.269,18.471,153.045
C05209=1084.845,-40.320,-55.202,174.271,18.472,153.045
C05210=1084.851,-40.070,-55.214,174.272,18.474,153.045
C05211=1084.857,-39.821,-55.227,174.274,18.475,153.045
C05212=1084.863,-39.571,-55.239,174.275,18.477,153.045
C05213=1084.869,-39.321,-55.251,174.277,18.480,153.045
C05214=1084.875,-39.072,-55.263,174.278,18.481,153.045
C05215=1084.880,-38.822,-55.276,174.280,18.483,153.045
C05216=1084.887,-38.572,-55.288,174.281,18.484,153.045
C05217=1084.892,-38.323,-55.300,174.283,18.486,153.045
C05218=1084.898,-38.073,-55.313,174.284,18.487,153.045
C05219=1084.904,-37.824,-55.325,174.285,18.489,153.046
C05220=1084.910,-37.574,-55.338,174.288,18.491,153.046
C05221=1084.916,-37.325,-55.349,174.289,18.493,153.046
C05222=1084.922,-37.075,-55.362,174.290,18.495,153.046
C05223=1084.928,-36.825,-55.374,174.292,18.496,153.046
C05224=1084.933,-36.576,-55.387,174.293,18.498,153.046
C05225=1084.939,-36.326,-55.399,174.294,18.500,153.046
C05226=1084.945,-36.076,-55.412,174.296,18.501,153.046
C05227=1084.951,-35.826,-55.424,174.298,18.503,153.046
C05228=1084.957,-35.577,-55.436,174.300,18.505,153.046
C05229=1084.963,-35.327,-55.448,174.301,18.507,153.046
C05230=1084.969,-35.078,-55.461,174.302,18.508,153.046
C05231=1084.975,-34.828,-55.473,174.304,18.510,153.046
C05232=1084.980,-34.578,-55.486,174.305,18.512,153.046
C05233=1084.986,-34.329,-55.498,174.306,18.514,153.046
C05234=1084.992,-34.079,-55.511,174.308,18.516,153.046
C05235=1084.998,-33.829,-55.524,174.310,18.517,153.047
C05236=1085.004,-33.581,-55.536,174.311,18.519,153.047
C05237=1085.010,-33.308,-55.550,174.312,18.521,153.047
C05238=1085.017,-33.036,-55.563,174.315,18.523,153.047
C05239=1085.024,-32.764,-55.577,174.316,18.524,153.047
C05240=1085.029,-32.492,-55.591,174.317,18.526,153.047
C05241=1085.036,-32.242,-55.603,174.319,18.528,153.047
C05242=1085.042,-31.992,-55.615,174.321,18.530,153.047
C05243=1085.048,-31.743,-55.628,174.322,18.532,153.047
C05244=1085.054,-31.493,-55.640,174.324,18.533,153.047
C05245=1085.059,-31.244,-55.652,174.325,18.535,153.047
C05246=1085.065,-30.994,-55.666,174.326,18.537,153.047
C05247=1085.071,-30.744,-55.678,174.328,18.538,153.047
C05248=1085.077,-30.495,-55.691,174.330,18.540,153.047
C05249=1085.083,-30.245,-55.703,174.331,18.542,153.047
C05250=1085.089,-29.995,-55.716,174.333,18.544,153.048
C05251=1085.094,-29.746,-55.729,174.334,18.546,153.048
C05252=1085.100,-29.496,-55.741,174.336,18.547,153.048
C05253=1085.106,-29.246,-55.754,174.337,18.549,153.048
C05254=1085.112,-28.997,-55.767,174.339,18.551,153.048
C05255=1085.119,-28.748,-55.779,174.340,18.553,153.048
C05256=1085.125,-28.498,-55.792,174.342,18.554,153.048
C05257=1085.130,-28.249,-55.804,174.343,18.556,153.048
C05258=1085.136,-27.999,-55.817,174.344,18.558,153.048
C05259=1085.142,-27.749,-55.830,174.346,18.559,153.048
C05260=1085.148,-27.499,-55.842,174.348,18.561,153.048
C05261=1085.154,-27.250,-55.855,174.350,18.563,153.048
C05262=1085.160,-27.000,-55.868,174.351,18.565,153.048
C05263=1085.166,-26.750,-55.881,174.352,18.567,153.048
C05264=1085.172,-26.501,-55.893,174.354,18.568,153.048
C05265=1085.178,-26.251,-55.905,174.356,18.571,153.049
C05266=1085.183,-26.002,-55.919,174.357,18.572,153.049
C05267=1085.189,-25.752,-55.932,174.358,18.574,153.049
C05268=1085.195,-25.502,-55.944,174.360,18.576,153.049
C05269=1085.201,-25.253,-55.958,174.361,18.577,153.049
C05270=1085.207,-25.003,-55.970,174.362,18.579,153.049
C05271=1085.213,-24.754,-55.983,174.365,18.581,153.049
C05272=1085.218,-24.504,-55.996,174.366,18.583,153.049
C05273=1085.224,-24.254,-56.009,174.367,18.585,153.049
C05274=1085.230,-24.005,-56.022,174.369,18.586,153.049
C05275=1085.236,-23.755,-56.035,174.370,18.588,153.049
C05276=1085.242,-23.505,-56.047,174.372,18.590,153.049
C05277=1085.248,-23.256,-56.060,174.374,18.592,153.049
C05278=1085.254,-23.006,-56.073,174.375,18.594,153.050
C05279=1085.259,-22.757,-56.087,174.376,18.595,153.050
C05280=1085.265,-22.507,-56.099,174.378,18.597,153.050
C05281=1085.271,-22.258,-56.112,174.380,18.600,153.050
C05282=1085.277,-22.008,-56.125,174.381,18.601,153.050
C05283=1085.283,-21.758,-56.137,174.382,18.603,153.050
C05284=1085.289,-21.509,-56.151,174.384,18.605,153.050
C05285=1085.294,-21.259,-56.164,174.385,18.606,153.050
C05286=1085.300,-21.010,-56.177,174.387,18.608,153.050
C05287=1085.306,-20.760,-56.190,174.389,18.610,153.050
C05288=1085.312,-20.510,-56.203,174.390,18.612,153.050
C05289=1085.318,-20.261,-56.216,174.391,18.613,153.050
C05290=1085.324,-20.011,-56.229,174.393,18.616,153.051
C05291=1085.329,-19.762,-56.242,174.395,18.618,153.051
C05292=1085.335,-19.513,-56.255,174.396,18.619,153.051
C05293=1085.341,-19.263,-56.267,174.397,18.621,153.051
C05294=1085.347,-19.013,-56.281,174.399,18.623,153.051
C05295=1085.353,-18.763,-56.294,174.400,18.624,153.051
C05296=1085.359,-18.514,-56.307,174.402,18.627,153.051
C05297=1085.365,-18.264,-56.320,174.404,18.628,153.051
C05298=1085.371,-18.015,-56.333,174.405,18.630,153.051
C05299=1085.376,-17.765,-56.347,174.407,18.631,153.051
C05300=1085.382,-17.515,-56.359,174.408,18.633,153.051
C05301=1085.389,-17.242,-56.374,174.410,18.636,153.051
C05302=1085.395,-16.969,-56.388,174.411,18.638,153.051
C05303=1085.401,-16.697,-56.402,174.413,18.640,153.051
C05304=1085.408,-16.423,-56.417,174.415,18.642,153.052
C05305=1085.414,-16.174,-56.430,174.416,18.643,153.052
C05306=1085.420,-15.924,-56.443,174.417,18.645,153.052
C05307=1085.426,-15.675,-56.456,174.419,18.647,153.052
C05308=1085.432,-15.425,-56.470,174.421,18.649,153.052
C05309=1085.438,-15.175,-56.483,174.422,18.650,153.052
C05310=1085.444,-14.926,-56.496,174.424,18.653,153.052
C05311=1085.450,-14.677,-56.510,174.426,18.655,153.052
C05312=1085.455,-14.427,-56.522,174.427,18.656,153.052
C05313=1085.462,-14.177,-56.536,174.428,18.658,153.052
C05314=1085.467,-13.928,-56.549,174.430,18.660,153.052
C05315=1085.473,-13.678,-56.562,174.431,18.661,153.052
C05316=1085.479,-13.428,-56.576,174.433,18.664,153.053
C05317=1085.485,-13.179,-56.589,174.435,18.665,153.053
C05318=1085.490,-12.929,-56.602,174.436,18.667,153.053
C05319=1085.496,-12.680,-56.616,174.437,18.669,153.053
C05320=1085.502,-12.430,-56.629,174.440,18.671,153.053
C05321=1085.508,-12.180,-56.642,174.441,18.673,153.053
C05322=1085.514,-11.931,-56.655,174.442,18.675,153.053
C05323=1085.519,-11.681,-56.669,174.443,18.677,153.053
C05324=1085.525,-11.432,-56.682,174.445,18.678,153.053
C05325=1085.531,-11.182,-56.695,174.447,18.680,153.053
C05326=1085.537,-10.933,-56.709,174.448,18.682,153.053
C05327=1085.542,-10.683,-56.723,174.450,18.684,153.053
C05328=1085.549,-10.434,-56.736,174.451,18.686,153.054
C05329=1085.555,-10.184,-56.749,174.453,18.688,153.054
C05330=1085.560,-9.934,-56.762,174.455,18.689,153.054
C05331=1085.566,-9.685,-56.776,174.456,18.692,153.054
C05332=1085.572,-9.435,-56.789,174.457,18.693,153.054
C05333=1085.578,-9.186,-56.803,174.459,18.696,153.054
C05334=1085.583,-8.937,-56.817,174.461,18.697,153.054
C05335=1085.589,-8.687,-56.829,174.462,18.699,153.054
C05336=1085.595,-8.437,-56.843,174.463,18.701,153.054
C05337=1085.601,-8.188,-56.856,174.465,18.703,153.054
C05338=1085.607,-7.938,-56.870,174.467,18.704,153.054
C05339=1085.613,-7.688,-56.884,174.468,18.706,153.055
C05340=1085.619,-7.439,-56.898,174.469,18.708,153.055
C05341=1085.625,-7.190,-56.911,174.471,18.710,153.055
C05342=1085.630,-6.939,-56.924,174.473,18.712,153.055
C05343=1085.636,-6.690,-56.937,174.474,18.714,153.055
C05344=1085.642,-6.440,-56.951,174.476,18.716,153.055
C05345=1085.648,-6.191,-56.964,174.477,18.717,153.055
C05346=1085.653,-5.942,-56.978,174.479,18.719,153.055
C05347=1085.660,-5.692,-56.992,174.480,18.721,153.055
C05348=1085.666,-5.442,-57.006,174.482,18.723,153.055
C05349=1085.672,-5.193,-57.019,174.483,18.725,153.055
C05350=1085.677,-4.943,-57.033,174.485,18.727,153.055
C05351=1085.683,-4.694,-57.047,174.487,18.728,153.055
C05352=1085.689,-4.444,-57.060,174.488,18.731,153.056
C05353=1085.695,-4.195,-57.074,174.489,18.732,153.056
C05354=1085.701,-3.945,-57.088,174.492,18.734,153.056
C05355=1085.707,-3.695,-57.101,174.493,18.736,153.056
C05356=1085.713,-3.446,-57.115,174.494,18.738,153.056
C05357=1085.719,-3.196,-57.129,174.495,18.740,153.056
C05358=1085.724,-2.947,-57.142,174.498,18.742,153.056
C05359=1085.730,-2.698,-57.156,174.499,18.743,153.056
C05360=1085.736,-2.448,-57.170,174.500,18.745,153.056
C05361=1085.741,-2.198,-57.183,174.502,18.747,153.056
C05362=1085.747,-1.949,-57.197,174.504,18.750,153.057
C05363=1085.753,-1.699,-57.211,174.505,18.751,153.057
C05364=1085.759,-1.449,-57.225,174.506,18.753,153.057
C05365=1085.765,-1.175,-57.239,174.509,18.755,153.057
C05366=1085.771,-0.901,-57.255,174.510,18.757,153.057
C05367=1085.778,-0.626,-57.270,174.512,18.760,153.057
C05368=1085.784,-0.351,-57.285,174.513,18.761,153.057
C05369=1085.790,-0.102,-57.299,174.514,18.763,153.057
C05370=1085.795,0.148,-57.313,174.517,18.765,153.057
C05371=1085.801,0.398,-57.327,174.518,18.767,153.057
C05372=1085.806,0.647,-57.341,174.519,18.769,153.058
C05373=1085.813,0.897,-57.354,174.521,18.772,153.058
C05374=1085.818,1.147,-57.368,174.523,18.773,153.058
C05375=1085.824,1.396,-57.383,174.524,18.775,153.058
C05376=1085.830,1.645,-57.397,174.525,18.777,153.058
C05377=1085.835,1.895,-57.411,174.528,18.779,153.058
C05378=1085.841,2.144,-57.424,174.529,18.781,153.058
C05379=1085.847,2.394,-57.438,174.530,18.782,153.058
C05380=1085.853,2.644,-57.452,174.531,18.784,153.058
C05381=1085.858,2.893,-57.466,174.534,18.786,153.058
C05382=1085.864,3.142,-57.480,174.535,18.788,153.059
C05383=1085.870,3.392,-57.494,174.536,18.790,153.059
C05384=1085.877,3.642,-57.508,174.539,18.792,153.059
C05385=1085.882,3.892,-57.522,174.540,18.794,153.059
C05386=1085.887,4.141,-57.536,174.541,18.796,153.059
C05387=1085.893,4.390,-57.550,174.542,18.798,153.059
C05388=1085.899,4.640,-57.564,174.545,18.800,153.059
C05389=1085.905,4.890,-57.578,174.546,18.802,153.059
C05390=1085.911,5.139,-57.592,174.547,18.803,153.059
C05391=1085.917,5.388,-57.606,174.549,18.805,153.059
C05392=1085.922,5.638,-57.620,174.551,18.807,153.059
C05393=1085.928,5.888,-57.634,174.552,18.809,153.059
C05394=1085.934,6.138,-57.648,174.553,18.811,153.060
C05395=1085.940,6.387,-57.663,174.556,18.813,153.060
C05396=1085.945,6.636,-57.677,174.557,18.815,153.060
C05397=1085.951,6.886,-57.691,174.558,18.817,153.060
C05398=1085.958,7.135,-57.705,174.560,18.818,153.060
C05399=1085.963,7.385,-57.719,174.562,18.821,153.060
C05400=1085.969,7.634,-57.732,174.563,18.822,153.060
C05401=1085.975,7.884,-57.747,174.564,18.824,153.060
C05402=1085.981,8.133,-57.761,174.567,18.826,153.060
C05403=1085.986,8.383,-57.775,174.568,18.828,153.060
C05404=1085.992,8.633,-57.790,174.569,18.830,153.060
C05405=1085.998,8.882,-57.804,174.571,18.831,153.061
C05406=1086.003,9.132,-57.818,174.573,18.834,153.061
C05407=1086.010,9.381,-57.832,174.574,18.836,153.061
C05408=1086.016,9.631,-57.846,174.576,18.837,153.061
C05409=1086.021,9.880,-57.860,174.578,18.840,153.061
C05410=1086.027,10.129,-57.874,174.579,18.841,153.061
C05411=1086.033,10.380,-57.889,174.580,18.843,153.061
C05412=1086.039,10.628,-57.903,174.582,18.845,153.061
C05413=1086.045,10.878,-57.917,174.584,18.847,153.061
C05414=1086.051,11.128,-57.931,174.585,18.849,153.061
C05415=1086.056,11.377,-57.946,174.587,18.850,153.061
C05416=1086.062,11.628,-57.960,174.589,18.852,153.061
C05417=1086.068,11.876,-57.975,174.590,18.854,153.062
C05418=1086.074,12.126,-57.989,174.591,18.856,153.062
C05419=1086.080,12.376,-58.004,174.593,18.859,153.062
C05420=1086.086,12.625,-58.017,174.595,18.860,153.062
C05421=1086.092,12.874,-58.031,174.596,18.862,153.062
C05422=1086.098,13.124,-58.046,174.598,18.864,153.062
C05423=1086.104,13.373,-58.060,174.600,18.866,153.062
C05424=1086.110,13.623,-58.074,174.601,18.867,153.062
C05425=1086.116,13.872,-58.089,174.602,18.869,153.062
C05426=1086.121,14.122,-58.103,174.605,18.871,153.062
C05427=1086.128,14.372,-58.118,174.606,18.873,153.062
C05428=1086.133,14.621,-58.132,174.607,18.875,153.062
C05429=1086.140,14.898,-58.148,174.609,18.877,153.063
C05430=1086.145,15.174,-58.164,174.611,18.879,153.063
C05431=1086.152,15.451,-58.181,174.613,18.882,153.063
C05432=1086.158,15.727,-58.196,174.614,18.883,153.063
C05433=1086.164,15.978,-58.211,174.616,18.886,153.063
C05434=1086.170,16.226,-58.225,174.618,18.887,153.063
C05435=1086.176,16.475,-58.240,174.619,18.889,153.063
C05436=1086.182,16.726,-58.254,174.621,18.891,153.063
C05437=1086.187,16.975,-58.269,174.623,18.893,153.063
C05438=1086.193,17.225,-58.283,174.624,18.895,153.063
C05439=1086.199,17.474,-58.298,174.626,18.897,153.063
C05440=1086.205,17.723,-58.313,174.627,18.899,153.064
C05441=1086.211,17.973,-58.327,174.629,18.900,153.064
C05442=1086.217,18.222,-58.341,174.631,18.903,153.064
C05443=1086.222,18.472,-58.357,174.632,18.905,153.064
C05444=1086.228,18.722,-58.371,174.634,18.906,153.064
C05445=1086.234,18.971,-58.385,174.636,18.909,153.064
C05446=1086.240,19.221,-58.400,174.637,18.910,153.064
C05447=1086.245,19.470,-58.414,174.638,18.912,153.064
C05448=1086.252,19.720,-58.429,174.641,18.914,153.064
C05449=1086.257,19.969,-58.444,174.642,18.916,153.064
C05450=1086.262,20.219,-58.458,174.643,18.918,153.065
C05451=1086.269,20.468,-58.473,174.645,18.920,153.065
C05452=1086.274,20.717,-58.488,174.647,18.921,153.065
